gfCNCPoint3[14451] = {X 398.8006, Y 41.5563, Z -4.6667, A 0.000, B 0.000, C 0.000 }
gfCNCPoint3[14452] = {X 399.4352, Y 40.8789, Z -4.6667, A 0.000, B 0.000, C 0.000 }
gfCNCPoint3[14453] = {X 399.4352, Y 31.6953, Z -4.6667, A 0.000, B 0.000, C 0.000 }
gfCNCPoint3[14454] = {X 393.4460, Y 21.2804, Z -4.6667, A 0.000, B 0.000, C 0.000 }
gfCNCPoint3[14455] = {X 392.5594, Y 19.7721, Z -4.6667, A 0.000, B 0.000, C 0.000 }
gfCNCPoint3[14456] = {X 391.6440, Y 18.2809, Z -4.6667, A 0.000, B 0.000, C 0.000 }
gfCNCPoint3[14457] = {X 391.1727, Y 17.6249, Z -4.6667, A 0.000, B 0.000, C 0.000 }
gfCNCPoint3[14458] = {X 390.6226, Y 17.0334, Z -4.6667, A 0.000, B 0.000, C 0.000 }
gfCNCPoint3[14459] = {X 389.8677, Y 16.6248, Z -4.6667, A 0.000, B 0.000, C 0.000 }
gfCNCPoint3[14460] = {X 389.2065, Y 16.0774, Z -4.6667, A 0.000, B 0.000, C 0.000 }
gfCNCPoint3[14461] = {X 388.6642, Y 15.4120, Z -4.6667, A 0.000, B 0.000, C 0.000 }
gfCNCPoint3[14462] = {X 388.2613, Y 14.6540, Z -4.6667, A 0.000, B 0.000, C 0.000 }
gfCNCPoint3[14463] = {X 388.0133, Y 13.8322, Z -4.6667, A 0.000, B 0.000, C 0.000 }
gfCNCPoint3[14464] = {X 387.9296, Y 12.9779, Z -4.6667, A 0.000, B 0.000, C 0.000 }
gfCNCPoint3[14465] = {X 387.9296, Y 12.1868, Z -4.6667, A 0.000, B 0.000, C 0.000 }
gfCNCPoint3[14466] = {X 388.0399, Y 11.2077, Z -4.6667, A 0.000, B 0.000, C 0.000 }
gfCNCPoint3[14467] = {X 388.3654, Y 10.2777, Z -4.6667, A 0.000, B 0.000, C 0.000 }
gfCNCPoint3[14468] = {X 388.8896, Y 9.4435, Z -4.6667, A 0.000, B 0.000, C 0.000 }
gfCNCPoint3[14469] = {X 389.5863, Y 8.7468, Z -4.6667, A 0.000, B 0.000, C 0.000 }
gfCNCPoint3[14470] = {X 390.4205, Y 8.2226, Z -4.6667, A 0.000, B 0.000, C 0.000 }
gfCNCPoint3[14471] = {X 391.3505, Y 7.8971, Z -4.6667, A 0.000, B 0.000, C 0.000 }
gfCNCPoint3[14472] = {X 392.3296, Y 7.7868, Z -4.6667, A 0.000, B 0.000, C 0.000 }
gfCNCPoint3[14473] = {X 399.1118, Y 7.7868, Z -4.6667, A 0.000, B 0.000, C 0.000 }
gfCNCPoint3[14474] = {X 400.0909, Y 7.8971, Z -4.6667, A 0.000, B 0.000, C 0.000 }
gfCNCPoint3[14475] = {X 401.0208, Y 8.2226, Z -4.6667, A 0.000, B 0.000, C 0.000 }
gfCNCPoint3[14476] = {X 401.8551, Y 8.7468, Z -4.6667, A 0.000, B 0.000, C 0.000 }
gfCNCPoint3[14477] = {X 402.5518, Y 9.4435, Z -4.6667, A 0.000, B 0.000, C 0.000 }
gfCNCPoint3[14478] = {X 403.0760, Y 10.2777, Z -4.6667, A 0.000, B 0.000, C 0.000 }
gfCNCPoint3[14479] = {X 403.4014, Y 11.2077, Z -4.6667, A 0.000, B 0.000, C 0.000 }
gfCNCPoint3[14480] = {X 403.5118, Y 12.1868, Z -4.6667, A 0.000, B 0.000, C 0.000 }
gfCNCPoint3[14481] = {X 403.5115, Y 13.0233, Z -4.6667, A 0.000, B 0.000, C 0.000 }
gfCNCPoint3[14482] = {X 403.4070, Y 13.9326, Z -4.6667, A 0.000, B 0.000, C 0.000 }
gfCNCPoint3[14483] = {X 403.1165, Y 14.8007, Z -4.6667, A 0.000, B 0.000, C 0.000 }
gfCNCPoint3[14484] = {X 405.3504, Y 18.6797, Z -4.6667, A 0.000, B 0.000, C 0.000 }
gfCNCPoint3[14485] = {X 407.7810, Y 14.7428, Z -4.6667, A 0.000, B 0.000, C 0.000 }
gfCNCPoint3[14486] = {X 407.5049, Y 13.8795, Z -4.6667, A 0.000, B 0.000, C 0.000 }
gfCNCPoint3[14487] = {X 407.4115, Y 12.9779, Z -4.6667, A 0.000, B 0.000, C 0.000 }
gfCNCPoint3[14488] = {X 407.4115, Y 12.1868, Z -4.6667, A 0.000, B 0.000, C 0.000 }
gfCNCPoint3[14489] = {X 407.5219, Y 11.2077, Z -4.6667, A 0.000, B 0.000, C 0.000 }
gfCNCPoint3[14490] = {X 407.8473, Y 10.2777, Z -4.6667, A 0.000, B 0.000, C 0.000 }
gfCNCPoint3[14491] = {X 408.3715, Y 9.4435, Z -4.6667, A 0.000, B 0.000, C 0.000 }
gfCNCPoint3[14492] = {X 409.0682, Y 8.7468, Z -4.6667, A 0.000, B 0.000, C 0.000 }
gfCNCPoint3[14493] = {X 409.9025, Y 8.2226, Z -4.6667, A 0.000, B 0.000, C 0.000 }
gfCNCPoint3[14494] = {X 410.8324, Y 7.8971, Z -4.6667, A 0.000, B 0.000, C 0.000 }
gfCNCPoint3[14495] = {X 411.8115, Y 7.7868, Z -4.6667, A 0.000, B 0.000, C 0.000 }
gfCNCPoint3[14496] = {X 419.3245, Y 7.7868, Z -4.6667, A 0.000, B 0.000, C 0.000 }
gfCNCPoint3[14497] = {X 420.3036, Y 7.8971, Z -4.6667, A 0.000, B 0.000, C 0.000 }
gfCNCPoint3[14498] = {X 421.2335, Y 8.2226, Z -4.6667, A 0.000, B 0.000, C 0.000 }
gfCNCPoint3[14499] = {X 422.0678, Y 8.7468, Z -4.6667, A 0.000, B 0.000, C 0.000 }
gfCNCPoint3[14500] = {X 422.7645, Y 9.4435, Z -4.6667, A 0.000, B 0.000, C 0.000 }
gfCNCPoint3[14501] = {X 423.2887, Y 10.2777, Z -4.6667, A 0.000, B 0.000, C 0.000 }
gfCNCPoint3[14502] = {X 423.6141, Y 11.2077, Z -4.6667, A 0.000, B 0.000, C 0.000 }
gfCNCPoint3[14503] = {X 423.7245, Y 12.1868, Z -4.6667, A 0.000, B 0.000, C 0.000 }
gfCNCPoint3[14504] = {X 423.7244, Y 12.9809, Z -4.6667, A 0.000, B 0.000, C 0.000 }
gfCNCPoint3[14505] = {X 423.6306, Y 13.8597, Z -4.6667, A 0.000, B 0.000, C 0.000 }
gfCNCPoint3[14506] = {X 423.3654, Y 14.7028, Z -4.6667, A 0.000, B 0.000, C 0.000 }
gfCNCPoint3[14507] = {X 422.9393, Y 15.4771, Z -4.6667, A 0.000, B 0.000, C 0.000 }
gfCNCPoint3[14508] = {X 422.3690, Y 16.1522, Z -4.6667, A 0.000, B 0.000, C 0.000 }
gfCNCPoint3[14509] = {X 421.6768, Y 16.7018, Z -4.6667, A 0.000, B 0.000, C 0.000 }
gfCNCPoint3[14510] = {X 420.8900, Y 17.1043, Z -4.6667, A 0.000, B 0.000, C 0.000 }
gfCNCPoint3[14511] = {X 420.1830, Y 18.0570, Z -4.6667, A 0.000, B 0.000, C 0.000 }
gfCNCPoint3[14512] = {X 419.5428, Y 19.0559, Z -4.6667, A 0.000, B 0.000, C 0.000 }
gfCNCPoint3[14513] = {X 418.0618, Y 21.4538, Z -4.6667, A 0.000, B 0.000, C 0.000 }
gfCNCPoint3[14514] = {X 411.6269, Y 31.7880, Z -4.6667, A 0.000, B 0.000, C 0.000 }
gfCNCPoint3[14515] = {X 411.6276, Y 40.8617, Z -4.6667, A 0.000, B 0.000, C 0.000 }
gfCNCPoint3[14516] = {X 412.2667, Y 41.5585, Z -4.6667, A 0.000, B 0.000, C 0.000 }
gfCNCPoint3[14517] = {X 412.7469, Y 42.3730, Z -4.6667, A 0.000, B 0.000, C 0.000 }
gfCNCPoint3[14518] = {X 413.0473, Y 43.2695, Z -4.6667, A 0.000, B 0.000, C 0.000 }
gfCNCPoint3[14519] = {X 413.1547, Y 44.2089, Z -4.6667, A 0.000, B 0.000, C 0.000 }
gfCNCPoint3[14520] = {X 413.1545, Y 45.0423, Z -4.6667, A 0.000, B 0.000, C 0.000 }
gfCNCPoint3[14521] = {X 413.0719, Y 45.8494, Z -4.6667, A 0.000, B 0.000, C 0.000 }
gfCNCPoint3[14522] = {X 412.8426, Y 46.6276, Z -4.6667, A 0.000, B 0.000, C 0.000 }
gfCNCPoint3[14523] = {X 412.4743, Y 47.3505, Z -4.6667, A 0.000, B 0.000, C 0.000 }
gfCNCPoint3[14524] = {X 411.9795, Y 47.9934, Z -4.6667, A 0.000, B 0.000, C 0.000 }
gfCNCPoint3[14525] = {X 412.3313, Y 48.3200, Z -4.6667, A 0.000, B 0.000, C 0.000 }
gfCNCPoint3[14526] = {X 419.4886, Y 48.3200, Z -4.6667, A 0.000, B 0.000, C 0.000 }
gfCNCPoint3[14527] = {X 420.8006, Y 48.4093, Z -4.6667, A 0.000, B 0.000, C 0.000 }
gfCNCPoint3[14528] = {X 422.0883, Y 48.6756, Z -4.6667, A 0.000, B 0.000, C 0.000 }
gfCNCPoint3[14529] = {X 423.3281, Y 49.1140, Z -4.6667, A 0.000, B 0.000, C 0.000 }
gfCNCPoint3[14530] = {X 424.4970, Y 49.7164, Z -4.6667, A 0.000, B 0.000, C 0.000 }
gfCNCPoint3[14531] = {X 425.4625, Y 50.3832, Z -4.6667, A 0.000, B 0.000, C 0.000 }
gfCNCPoint3[14532] = {X 426.3402, Y 51.1620, Z -4.6667, A 0.000, B 0.000, C 0.000 }
gfCNCPoint3[14533] = {X 427.1172, Y 52.0412, Z -4.6667, A 0.000, B 0.000, C 0.000 }
gfCNCPoint3[14534] = {X 427.7821, Y 53.0080, Z -4.6667, A 0.000, B 0.000, C 0.000 }
gfCNCPoint3[14535] = {X 428.1267, Y 53.6313, Z -4.6667, A 0.000, B 0.000, C 0.000 }
gfCNCPoint3[14536] = {X 428.4245, Y 54.2783, Z -4.6667, A 0.000, B 0.000, C 0.000 }
gfCNCPoint3[14537] = {X 431.5824, Y 55.5088, Z -4.6667, A 0.000, B 0.000, C 0.000 }
gfCNCPoint3[14538] = {X 449.5095, Y 62.6216, Z -4.6667, A 0.000, B 0.000, C 0.000 }
gfCNCPoint3[14539] = {X 449.1114, Y 61.4466, Z -4.6667, A 0.000, B 0.000, C 0.000 }
gfCNCPoint3[14540] = {X 448.8668, Y 60.2305, Z -4.6667, A 0.000, B 0.000, C 0.000 }
gfCNCPoint3[14541] = {X 448.7798, Y 58.9930, Z -4.6667, A 0.000, B 0.000, C 0.000 }
gfCNCPoint3[14542] = {X 448.7796, Y 58.0000, Z -4.6667, A 0.000, B 0.000, C 0.000 }
gfCNCPoint3[14543] = {X 448.8564, Y 56.7833, Z -4.6667, A 0.000, B 0.000, C 0.000 }
gfCNCPoint3[14544] = {X 449.0855, Y 55.5859, Z -4.6667, A 0.000, B 0.000, C 0.000 }
gfCNCPoint3[14545] = {X 449.4632, Y 54.4268, Z -4.6667, A 0.000, B 0.000, C 0.000 }
gfCNCPoint3[14546] = {X 449.9837, Y 53.3244, Z -4.6667, A 0.000, B 0.000, C 0.000 }
gfCNCPoint3[14547] = {X 450.6386, Y 52.2961, Z -4.6667, A 0.000, B 0.000, C 0.000 }
gfCNCPoint3[14548] = {X 451.3887, Y 51.3890, Z -4.6667, A 0.000, B 0.000, C 0.000 }
gfCNCPoint3[14549] = {X 452.2434, Y 50.5796, Z -4.6667, A 0.000, B 0.000, C 0.000 }
gfCNCPoint3[14550] = {X 453.1901, Y 49.8800, Z -4.6667, A 0.000, B 0.000, C 0.000 }
gfCNCPoint3[14551] = {X 452.3731, Y 49.8442, Z -4.6667, A 0.000, B 0.000, C 0.000 }
gfCNCPoint3[14552] = {X 451.5735, Y 49.6724, Z -4.6667, A 0.000, B 0.000, C 0.000 }
gfCNCPoint3[14553] = {X 450.8138, Y 49.3696, Z -4.6667, A 0.000, B 0.000, C 0.000 }
gfCNCPoint3[14554] = {X 450.1154, Y 48.9441, Z -4.6667, A 0.000, B 0.000, C 0.000 }
gfCNCPoint3[14555] = {X 449.3503, Y 48.2496, Z -4.6667, A 0.000, B 0.000, C 0.000 }
gfCNCPoint3[14556] = {X 448.7486, Y 47.4095, Z -4.6667, A 0.000, B 0.000, C 0.000 }
gfCNCPoint3[14557] = {X 448.3373, Y 46.4616, Z -4.6667, A 0.000, B 0.000, C 0.000 }
gfCNCPoint3[14558] = {X 448.1732, Y 45.7588, Z -4.6667, A 0.000, B 0.000, C 0.000 }
gfCNCPoint3[14559] = {X 448.1146, Y 45.0395, Z -4.6667, A 0.000, B 0.000, C 0.000 }
gfCNCPoint3[14560] = {X 448.1149, Y 44.1417, Z -4.6667, A 0.000, B 0.000, C 0.000 }
gfCNCPoint3[14561] = {X 448.2252, Y 43.1751, Z -4.6667, A 0.000, B 0.000, C 0.000 }
gfCNCPoint3[14562] = {X 448.5250, Y 42.2497, Z -4.6667, A 0.000, B 0.000, C 0.000 }
gfCNCPoint3[14563] = {X 449.0024, Y 41.4021, Z -4.6667, A 0.000, B 0.000, C 0.000 }
gfCNCPoint3[14564] = {X 449.6384, Y 40.6660, Z -4.6667, A 0.000, B 0.000, C 0.000 }
gfCNCPoint3[14565] = {X 449.6384, Y 35.0338, Z -4.6667, A 0.000, B 0.000, C 0.000 }
gfCNCPoint3[14566] = {X 447.8166, Y 35.0338, Z -4.6667, A 0.000, B 0.000, C 0.000 }
gfCNCPoint3[14567] = {X 444.1904, Y 42.0943, Z -4.6667, A 0.000, B 0.000, C 0.000 }
gfCNCPoint3[14568] = {X 443.7927, Y 42.8683, Z -4.6667, A 0.000, B 0.000, C 0.000 }
gfCNCPoint3[14569] = {X 443.9302, Y 43.5105, Z -4.6667, A 0.000, B 0.000, C 0.000 }
gfCNCPoint3[14570] = {X 443.9803, Y 44.1653, Z -4.6667, A 0.000, B 0.000, C 0.000 }
gfCNCPoint3[14571] = {X 443.9805, Y 45.0000, Z -4.6667, A 0.000, B 0.000, C 0.000 }
gfCNCPoint3[14572] = {X 443.9242, Y 45.7387, Z -4.6667, A 0.000, B 0.000, C 0.000 }
gfCNCPoint3[14573] = {X 443.7568, Y 46.4603, Z -4.6667, A 0.000, B 0.000, C 0.000 }
gfCNCPoint3[14574] = {X 443.3737, Y 47.3567, Z -4.6667, A 0.000, B 0.000, C 0.000 }
gfCNCPoint3[14575] = {X 442.8199, Y 48.1591, Z -4.6667, A 0.000, B 0.000, C 0.000 }
gfCNCPoint3[14576] = {X 442.1178, Y 48.8354, Z -4.6667, A 0.000, B 0.000, C 0.000 }
gfCNCPoint3[14577] = {X 441.2952, Y 49.3586, Z -4.6667, A 0.000, B 0.000, C 0.000 }
gfCNCPoint3[14578] = {X 440.3850, Y 49.7079, Z -4.6667, A 0.000, B 0.000, C 0.000 }
gfCNCPoint3[14579] = {X 441.6485, Y 54.3386, Z -4.6667, A 0.000, B 0.000, C 0.000 }
gfCNCPoint3[14580] = {X 444.2223, Y 55.3598, Z -4.6667, A 0.000, B 0.000, C 0.000 }
gfCNCPoint3[14581] = {X 444.5426, Y 54.0016, Z -4.6667, A 0.000, B 0.000, C 0.000 }
gfCNCPoint3[14582] = {X 444.9921, Y 52.6806, Z -4.6667, A 0.000, B 0.000, C 0.000 }
gfCNCPoint3[14583] = {X 443.9523, Y 53.3763, Z -4.6667, A 0.000, B 0.000, C 0.000 }
gfCNCPoint3[14584] = {X 442.8316, Y 53.9320, Z -4.6667, A 0.000, B 0.000, C 0.000 }
gfCNCPoint3[14585] = {X 441.6485, Y 54.3386, Z -4.6667, A 0.000, B 0.000, C 0.000 }
gfCNCPoint3[14586] = {X 441.0167, Y 52.0233, Z -4.6667, A 0.000, B 0.000, C 0.000 }
gfCNCPoint3[14587] = {X 440.0672, Y 52.2155, Z -4.6667, A 0.000, B 0.000, C 0.000 }
gfCNCPoint3[14588] = {X 439.1005, Y 52.2800, Z -4.6667, A 0.000, B 0.000, C 0.000 }
gfCNCPoint3[14589] = {X 432.5144, Y 52.2800, Z -4.6667, A 0.000, B 0.000, C 0.000 }
gfCNCPoint3[14590] = {X 431.6034, Y 52.2228, Z -4.6667, A 0.000, B 0.000, C 0.000 }
gfCNCPoint3[14591] = {X 430.7067, Y 52.0520, Z -4.6667, A 0.000, B 0.000, C 0.000 }
gfCNCPoint3[14592] = {X 429.8384, Y 51.7703, Z -4.6667, A 0.000, B 0.000, C 0.000 }
gfCNCPoint3[14593] = {X 430.0169, Y 52.0771, Z -4.6667, A 0.000, B 0.000, C 0.000 }
gfCNCPoint3[14594] = {X 430.1864, Y 52.3890, Z -4.6667, A 0.000, B 0.000, C 0.000 }
gfCNCPoint3[14595] = {X 432.4641, Y 53.2767, Z -4.6667, A 0.000, B 0.000, C 0.000 }
gfCNCPoint3[14596] = {X 446.3797, Y 58.7978, Z -4.6667, A 0.000, B 0.000, C 0.000 }
gfCNCPoint3[14597] = {X 446.3796, Y 58.0000, Z -4.6667, A 0.000, B 0.000, C 0.000 }
gfCNCPoint3[14598] = {X 446.4303, Y 56.8941, Z -4.6667, A 0.000, B 0.000, C 0.000 }
gfCNCPoint3[14599] = {X 446.5821, Y 55.7974, Z -4.6667, A 0.000, B 0.000, C 0.000 }
gfCNCPoint3[14600] = {X 446.8493, Y 54.6644, Z -4.6667, A 0.000, B 0.000, C 0.000 }
gfCNCPoint3[14601] = {X 447.2243, Y 53.5622, Z -4.6667, A 0.000, B 0.000, C 0.000 }
gfCNCPoint3[14602] = {X 447.8767, Y 52.1752, Z -4.6667, A 0.000, B 0.000, C 0.000 }
gfCNCPoint3[14603] = {X 448.6995, Y 50.8820, Z -4.6667, A 0.000, B 0.000, C 0.000 }
gfCNCPoint3[14604] = {X 447.8224, Y 50.1272, Z -4.6667, A 0.000, B 0.000, C 0.000 }
gfCNCPoint3[14605] = {X 447.0760, Y 49.2431, Z -4.6667, A 0.000, B 0.000, C 0.000 }
gfCNCPoint3[14606] = {X 446.4792, Y 48.2518, Z -4.6667, A 0.000, B 0.000, C 0.000 }
gfCNCPoint3[14607] = {X 446.0469, Y 47.1785, Z -4.6667, A 0.000, B 0.000, C 0.000 }
gfCNCPoint3[14608] = {X 445.6333, Y 48.2126, Z -4.6667, A 0.000, B 0.000, C 0.000 }
gfCNCPoint3[14609] = {X 445.0668, Y 49.1715, Z -4.6667, A 0.000, B 0.000, C 0.000 }
gfCNCPoint3[14610] = {X 444.3606, Y 50.0328, Z -4.6667, A 0.000, B 0.000, C 0.000 }
gfCNCPoint3[14611] = {X 443.5314, Y 50.7763, Z -4.6667, A 0.000, B 0.000, C 0.000 }
gfCNCPoint3[14612] = {X 442.7494, Y 51.2995, Z -4.6667, A 0.000, B 0.000, C 0.000 }
gfCNCPoint3[14613] = {X 441.9065, Y 51.7175, Z -4.6667, A 0.000, B 0.000, C 0.000 }
gfCNCPoint3[14614] = {X 441.0167, Y 52.0233, Z -4.6667, A 0.000, B 0.000, C 0.000 }
gfCNCPoint3[14615] = {X 440.3850, Y 49.7079, Z -4.6667, A 0.000, B 0.000, C 0.000 }
gfCNCPoint3[14616] = {X 439.7485, Y 49.8368, Z -4.6667, A 0.000, B 0.000, C 0.000 }
gfCNCPoint3[14617] = {X 439.1005, Y 49.8800, Z -4.6667, A 0.000, B 0.000, C 0.000 }
gfCNCPoint3[14618] = {X 432.5144, Y 49.8800, Z -4.6667, A 0.000, B 0.000, C 0.000 }
gfCNCPoint3[14619] = {X 431.6014, Y 49.7938, Z -4.6667, A 0.000, B 0.000, C 0.000 }
gfCNCPoint3[14620] = {X 430.7206, Y 49.5383, Z -4.6667, A 0.000, B 0.000, C 0.000 }
gfCNCPoint3[14621] = {X 429.8343, Y 49.0782, Z -4.6667, A 0.000, B 0.000, C 0.000 }
gfCNCPoint3[14622] = {X 429.0603, Y 48.4473, Z -4.6667, A 0.000, B 0.000, C 0.000 }
gfCNCPoint3[14623] = {X 428.4309, Y 47.6720, Z -4.6667, A 0.000, B 0.000, C 0.000 }
gfCNCPoint3[14624] = {X 427.9725, Y 46.7848, Z -4.6667, A 0.000, B 0.000, C 0.000 }
gfCNCPoint3[14625] = {X 427.7197, Y 45.9083, Z -4.6667, A 0.000, B 0.000, C 0.000 }
gfCNCPoint3[14626] = {X 427.6344, Y 45.0000, Z -4.6667, A 0.000, B 0.000, C 0.000 }
gfCNCPoint3[14627] = {X 427.6344, Y 44.2089, Z -4.6667, A 0.000, B 0.000, C 0.000 }
gfCNCPoint3[14628] = {X 427.7263, Y 43.2661, Z -4.6667, A 0.000, B 0.000, C 0.000 }
gfCNCPoint3[14629] = {X 427.9987, Y 42.3588, Z -4.6667, A 0.000, B 0.000, C 0.000 }
gfCNCPoint3[14630] = {X 428.4411, Y 41.5212, Z -4.6667, A 0.000, B 0.000, C 0.000 }
gfCNCPoint3[14631] = {X 429.0371, Y 40.7849, Z -4.6667, A 0.000, B 0.000, C 0.000 }
gfCNCPoint3[14632] = {X 429.7641, Y 40.1776, Z -4.6667, A 0.000, B 0.000, C 0.000 }
gfCNCPoint3[14633] = {X 430.5947, Y 39.7222, Z -4.6667, A 0.000, B 0.000, C 0.000 }
gfCNCPoint3[14634] = {X 434.2537, Y 32.5603, Z -4.6667, A 0.000, B 0.000, C 0.000 }
gfCNCPoint3[14635] = {X 433.1657, Y 31.7642, Z -4.6667, A 0.000, B 0.000, C 0.000 }
gfCNCPoint3[14636] = {X 432.1744, Y 30.8506, Z -4.6667, A 0.000, B 0.000, C 0.000 }
gfCNCPoint3[14637] = {X 431.2923, Y 29.8311, Z -4.6667, A 0.000, B 0.000, C 0.000 }
gfCNCPoint3[14638] = {X 430.5307, Y 28.7187, Z -4.6667, A 0.000, B 0.000, C 0.000 }
gfCNCPoint3[14639] = {X 422.3160, Y 33.6865, Z -4.6667, A 0.000, B 0.000, C 0.000 }
gfCNCPoint3[14640] = {X 421.8924, Y 34.3679, Z -4.6667, A 0.000, B 0.000, C 0.000 }
gfCNCPoint3[14641] = {X 422.1472, Y 34.0999, Z -4.6667, A 0.000, B 0.000, C 0.000 }
gfCNCPoint3[14642] = {X 422.4087, Y 33.8384, Z -4.6667, A 0.000, B 0.000, C 0.000 }
gfCNCPoint3[14643] = {X 422.3622, Y 33.7626, Z -4.6667, A 0.000, B 0.000, C 0.000 }
gfCNCPoint3[14644] = {X 422.3160, Y 33.6865, Z -4.6667, A 0.000, B 0.000, C 0.000 }
gfCNCPoint3[14645] = {X 424.3697, Y 32.4446, Z -4.6667, A 0.000, B 0.000, C 0.000 }
gfCNCPoint3[14646] = {X 423.3882, Y 30.6017, Z -4.6667, A 0.000, B 0.000, C 0.000 }
gfCNCPoint3[14647] = {X 422.6133, Y 28.6629, Z -4.6667, A 0.000, B 0.000, C 0.000 }
gfCNCPoint3[14648] = {X 419.3071, Y 33.9807, Z -4.6667, A 0.000, B 0.000, C 0.000 }
gfCNCPoint3[14649] = {X 419.3074, Y 38.3388, Z -4.6667, A 0.000, B 0.000, C 0.000 }
gfCNCPoint3[14650] = {X 419.9578, Y 39.7076, Z -4.6667, A 0.000, B 0.000, C 0.000 }
gfCNCPoint3[14651] = {X 420.4336, Y 41.1465, Z -4.6667, A 0.000, B 0.000, C 0.000 }
gfCNCPoint3[14652] = {X 420.6279, Y 41.1585, Z -4.6667, A 0.000, B 0.000, C 0.000 }
gfCNCPoint3[14653] = {X 420.8222, Y 41.1728, Z -4.6667, A 0.000, B 0.000, C 0.000 }
gfCNCPoint3[14654] = {X 421.2843, Y 39.7578, Z -4.6667, A 0.000, B 0.000, C 0.000 }
gfCNCPoint3[14655] = {X 421.9170, Y 38.4105, Z -4.6667, A 0.000, B 0.000, C 0.000 }
gfCNCPoint3[14656] = {X 422.7105, Y 37.1511, Z -4.6667, A 0.000, B 0.000, C 0.000 }
gfCNCPoint3[14657] = {X 423.6530, Y 35.9990, Z -4.6667, A 0.000, B 0.000, C 0.000 }
gfCNCPoint3[14658] = {X 424.3415, Y 35.3133, Z -4.6667, A 0.000, B 0.000, C 0.000 }
gfCNCPoint3[14659] = {X 425.0829, Y 34.6852, Z -4.6667, A 0.000, B 0.000, C 0.000 }
gfCNCPoint3[14660] = {X 425.4267, Y 34.0121, Z -4.6667, A 0.000, B 0.000, C 0.000 }
gfCNCPoint3[14661] = {X 424.8788, Y 33.2414, Z -4.6667, A 0.000, B 0.000, C 0.000 }
gfCNCPoint3[14662] = {X 424.3697, Y 32.4446, Z -4.6667, A 0.000, B 0.000, C 0.000 }
gfCNCPoint3[14663] = {X 426.4233, Y 31.2026, Z -4.6667, A 0.000, B 0.000, C 0.000 }
gfCNCPoint3[14664] = {X 425.5649, Y 29.5907, Z -4.6667, A 0.000, B 0.000, C 0.000 }
gfCNCPoint3[14665] = {X 424.8871, Y 27.8950, Z -4.6667, A 0.000, B 0.000, C 0.000 }
gfCNCPoint3[14666] = {X 424.6543, Y 27.1484, Z -4.6667, A 0.000, B 0.000, C 0.000 }
gfCNCPoint3[14667] = {X 424.4565, Y 26.3919, Z -4.6667, A 0.000, B 0.000, C 0.000 }
gfCNCPoint3[14668] = {X 424.0556, Y 24.2623, Z -4.6667, A 0.000, B 0.000, C 0.000 }
gfCNCPoint3[14669] = {X 423.8652, Y 22.1037, Z -4.6667, A 0.000, B 0.000, C 0.000 }
gfCNCPoint3[14670] = {X 416.9071, Y 33.2955, Z -4.6667, A 0.000, B 0.000, C 0.000 }
gfCNCPoint3[14671] = {X 416.9075, Y 38.9954, Z -4.6667, A 0.000, B 0.000, C 0.000 }
gfCNCPoint3[14672] = {X 417.4888, Y 40.0487, Z -4.6667, A 0.000, B 0.000, C 0.000 }
gfCNCPoint3[14673] = {X 417.9368, Y 41.1651, Z -4.6667, A 0.000, B 0.000, C 0.000 }
gfCNCPoint3[14674] = {X 418.2446, Y 42.3281, Z -4.6667, A 0.000, B 0.000, C 0.000 }
gfCNCPoint3[14675] = {X 418.4076, Y 43.5200, Z -4.6667, A 0.000, B 0.000, C 0.000 }
gfCNCPoint3[14676] = {X 419.4886, Y 43.5200, Z -4.6667, A 0.000, B 0.000, C 0.000 }
gfCNCPoint3[14677] = {X 421.1752, Y 43.6186, Z -4.6667, A 0.000, B 0.000, C 0.000 }
gfCNCPoint3[14678] = {X 422.8389, Y 43.9129, Z -4.6667, A 0.000, B 0.000, C 0.000 }
gfCNCPoint3[14679] = {X 423.0005, Y 42.4234, Z -4.6667, A 0.000, B 0.000, C 0.000 }
gfCNCPoint3[14680] = {X 423.3900, Y 40.9766, Z -4.6667, A 0.000, B 0.000, C 0.000 }
gfCNCPoint3[14681] = {X 423.9980, Y 39.6073, Z -4.6667, A 0.000, B 0.000, C 0.000 }
gfCNCPoint3[14682] = {X 424.8102, Y 38.3482, Z -4.6667, A 0.000, B 0.000, C 0.000 }
gfCNCPoint3[14683] = {X 425.8068, Y 37.2295, Z -4.6667, A 0.000, B 0.000, C 0.000 }
gfCNCPoint3[14684] = {X 426.9642, Y 36.2780, Z -4.6667, A 0.000, B 0.000, C 0.000 }
gfCNCPoint3[14685] = {X 428.2773, Y 33.7078, Z -4.6667, A 0.000, B 0.000, C 0.000 }
gfCNCPoint3[14686] = {X 427.2919, Y 32.4984, Z -4.6667, A 0.000, B 0.000, C 0.000 }
gfCNCPoint3[14687] = {X 426.4233, Y 31.2026, Z -4.6667, A 0.000, B 0.000, C 0.000 }
gfCNCPoint3[14688] = {X 428.4770, Y 29.9607, Z -4.6667, A 0.000, B 0.000, C 0.000 }
gfCNCPoint3[14689] = {X 427.7729, Y 28.6468, Z -4.6667, A 0.000, B 0.000, C 0.000 }
gfCNCPoint3[14690] = {X 427.2090, Y 27.2670, Z -4.6667, A 0.000, B 0.000, C 0.000 }
gfCNCPoint3[14691] = {X 426.7913, Y 25.8360, Z -4.6667, A 0.000, B 0.000, C 0.000 }
gfCNCPoint3[14692] = {X 426.4333, Y 23.9362, Z -4.6667, A 0.000, B 0.000, C 0.000 }
gfCNCPoint3[14693] = {X 426.2634, Y 22.0104, Z -4.6667, A 0.000, B 0.000, C 0.000 }
gfCNCPoint3[14694] = {X 426.2915, Y 19.9433, Z -4.6667, A 0.000, B 0.000, C 0.000 }
gfCNCPoint3[14695] = {X 426.5362, Y 17.8906, Z -4.6667, A 0.000, B 0.000, C 0.000 }
gfCNCPoint3[14696] = {X 426.9947, Y 15.8749, Z -4.6667, A 0.000, B 0.000, C 0.000 }
gfCNCPoint3[14697] = {X 427.6132, Y 14.1191, Z -4.6667, A 0.000, B 0.000, C 0.000 }
gfCNCPoint3[14698] = {X 428.4475, Y 12.4549, Z -4.6667, A 0.000, B 0.000, C 0.000 }
gfCNCPoint3[14699] = {X 429.4841, Y 10.9087, Z -4.6667, A 0.000, B 0.000, C 0.000 }
gfCNCPoint3[14700] = {X 430.7069, Y 9.5050, Z -4.6667, A 0.000, B 0.000, C 0.000 }
gfCNCPoint3[14701] = {X 426.0925, Y 9.5050, Z -4.6667, A 0.000, B 0.000, C 0.000 }
gfCNCPoint3[14702] = {X 426.3754, Y 10.3750, Z -4.6667, A 0.000, B 0.000, C 0.000 }
gfCNCPoint3[14703] = {X 426.5470, Y 11.2737, Z -4.6667, A 0.000, B 0.000, C 0.000 }
gfCNCPoint3[14704] = {X 426.6045, Y 12.1868, Z -4.6667, A 0.000, B 0.000, C 0.000 }
gfCNCPoint3[14705] = {X 426.6045, Y 12.9851, Z -4.6667, A 0.000, B 0.000, C 0.000 }
gfCNCPoint3[14706] = {X 426.4815, Y 14.2871, Z -4.6667, A 0.000, B 0.000, C 0.000 }
gfCNCPoint3[14707] = {X 426.1296, Y 15.5465, Z -4.6667, A 0.000, B 0.000, C 0.000 }
gfCNCPoint3[14708] = {X 425.5599, Y 16.7236, Z -4.6667, A 0.000, B 0.000, C 0.000 }
gfCNCPoint3[14709] = {X 424.7904, Y 17.7810, Z -4.6667, A 0.000, B 0.000, C 0.000 }
gfCNCPoint3[14710] = {X 423.8456, Y 18.6852, Z -4.6667, A 0.000, B 0.000, C 0.000 }
gfCNCPoint3[14711] = {X 422.7555, Y 19.4074, Z -4.6667, A 0.000, B 0.000, C 0.000 }
gfCNCPoint3[14712] = {X 422.3655, Y 19.9717, Z -4.6667, A 0.000, B 0.000, C 0.000 }
gfCNCPoint3[14713] = {X 422.0027, Y 20.5539, Z -4.6667, A 0.000, B 0.000, C 0.000 }
gfCNCPoint3[14714] = {X 414.5070, Y 32.6104, Z -4.6667, A 0.000, B 0.000, C 0.000 }
gfCNCPoint3[14715] = {X 414.5075, Y 39.7469, Z -4.6667, A 0.000, B 0.000, C 0.000 }
gfCNCPoint3[14716] = {X 415.1561, Y 40.7519, Z -4.6667, A 0.000, B 0.000, C 0.000 }
gfCNCPoint3[14717] = {X 415.6344, Y 41.8483, Z -4.6667, A 0.000, B 0.000, C 0.000 }
gfCNCPoint3[14718] = {X 415.9298, Y 43.0074, Z -4.6667, A 0.000, B 0.000, C 0.000 }
gfCNCPoint3[14719] = {X 416.0347, Y 44.1990, Z -4.6667, A 0.000, B 0.000, C 0.000 }
gfCNCPoint3[14720] = {X 416.0347, Y 44.9999, Z -4.6667, A 0.000, B 0.000, C 0.000 }
gfCNCPoint3[14721] = {X 416.0201, Y 45.4609, Z -4.6667, A 0.000, B 0.000, C 0.000 }
gfCNCPoint3[14722] = {X 415.9763, Y 45.9200, Z -4.6667, A 0.000, B 0.000, C 0.000 }
gfCNCPoint3[14723] = {X 419.4886, Y 45.9200, Z -4.6667, A 0.000, B 0.000, C 0.000 }
gfCNCPoint3[14724] = {X 420.8957, Y 46.0022, Z -4.6667, A 0.000, B 0.000, C 0.000 }
gfCNCPoint3[14725] = {X 422.2836, Y 46.2478, Z -4.6667, A 0.000, B 0.000, C 0.000 }
gfCNCPoint3[14726] = {X 423.4822, Y 46.5992, Z -4.6667, A 0.000, B 0.000, C 0.000 }
gfCNCPoint3[14727] = {X 424.6380, Y 47.0725, Z -4.6667, A 0.000, B 0.000, C 0.000 }
gfCNCPoint3[14728] = {X 425.7388, Y 47.6626, Z -4.6667, A 0.000, B 0.000, C 0.000 }
gfCNCPoint3[14729] = {X 425.4600, Y 46.7984, Z -4.6667, A 0.000, B 0.000, C 0.000 }
gfCNCPoint3[14730] = {X 425.2910, Y 45.9063, Z -4.6667, A 0.000, B 0.000, C 0.000 }
gfCNCPoint3[14731] = {X 425.2344, Y 45.0000, Z -4.6667, A 0.000, B 0.000, C 0.000 }
gfCNCPoint3[14732] = {X 425.2344, Y 44.2089, Z -4.6667, A 0.000, B 0.000, C 0.000 }
gfCNCPoint3[14733] = {X 425.2353, Y 44.0976, Z -4.6667, A 0.000, B 0.000, C 0.000 }
gfCNCPoint3[14734] = {X 425.2378, Y 43.9863, Z -4.6667, A 0.000, B 0.000, C 0.000 }
gfCNCPoint3[14735] = {X 425.3770, Y 42.7748, Z -4.6667, A 0.000, B 0.000, C 0.000 }
gfCNCPoint3[14736] = {X 425.7165, Y 41.6036, Z -4.6667, A 0.000, B 0.000, C 0.000 }
gfCNCPoint3[14737] = {X 426.2468, Y 40.5054, Z -4.6667, A 0.000, B 0.000, C 0.000 }
gfCNCPoint3[14738] = {X 426.9528, Y 39.5112, Z -4.6667, A 0.000, B 0.000, C 0.000 }
gfCNCPoint3[14739] = {X 427.8150, Y 38.6488, Z -4.6667, A 0.000, B 0.000, C 0.000 }
gfCNCPoint3[14740] = {X 428.8090, Y 37.9424, Z -4.6667, A 0.000, B 0.000, C 0.000 }
gfCNCPoint3[14741] = {X 431.2079, Y 33.2468, Z -4.6667, A 0.000, B 0.000, C 0.000 }
gfCNCPoint3[14742] = {X 430.1898, Y 32.2441, Z -4.6667, A 0.000, B 0.000, C 0.000 }
gfCNCPoint3[14743] = {X 429.2764, Y 31.1451, Z -4.6667, A 0.000, B 0.000, C 0.000 }
gfCNCPoint3[14744] = {X 428.4770, Y 29.9607, Z -4.6667, A 0.000, B 0.000, C 0.000 }
gfCNCPoint3[14745] = {X 430.5307, Y 28.7187, Z -4.6667, A 0.000, B 0.000, C 0.000 }
gfCNCPoint3[14746] = {X 429.9438, Y 27.6235, Z -4.6667, A 0.000, B 0.000, C 0.000 }
gfCNCPoint3[14747] = {X 429.4739, Y 26.4732, Z -4.6667, A 0.000, B 0.000, C 0.000 }
gfCNCPoint3[14748] = {X 429.1261, Y 25.2803, Z -4.6667, A 0.000, B 0.000, C 0.000 }
gfCNCPoint3[14749] = {X 428.8017, Y 23.5412, Z -4.6667, A 0.000, B 0.000, C 0.000 }
gfCNCPoint3[14750] = {X 428.6567, Y 21.7780, Z -4.6667, A 0.000, B 0.000, C 0.000 }
gfCNCPoint3[14751] = {X 428.6927, Y 20.0093, Z -4.6667, A 0.000, B 0.000, C 0.000 }
gfCNCPoint3[14752] = {X 428.9091, Y 18.2534, Z -4.6667, A 0.000, B 0.000, C 0.000 }
gfCNCPoint3[14753] = {X 429.3039, Y 16.5289, Z -4.6667, A 0.000, B 0.000, C 0.000 }
gfCNCPoint3[14754] = {X 429.8220, Y 15.0579, Z -4.6667, A 0.000, B 0.000, C 0.000 }
gfCNCPoint3[14755] = {X 430.5209, Y 13.6636, Z -4.6667, A 0.000, B 0.000, C 0.000 }
gfCNCPoint3[14756] = {X 431.3894, Y 12.3682, Z -4.6667, A 0.000, B 0.000, C 0.000 }
gfCNCPoint3[14757] = {X 432.4138, Y 11.1921, Z -4.6667, A 0.000, B 0.000, C 0.000 }
gfCNCPoint3[14758] = {X 433.5453, Y 10.1797, Z -4.6667, A 0.000, B 0.000, C 0.000 }
gfCNCPoint3[14759] = {X 434.7922, Y 9.3133, Z -4.6667, A 0.000, B 0.000, C 0.000 }
gfCNCPoint3[14760] = {X 436.1357, Y 8.6059, Z -4.6667, A 0.000, B 0.000, C 0.000 }
gfCNCPoint3[14761] = {X 437.5557, Y 8.0683, Z -4.6667, A 0.000, B 0.000, C 0.000 }
gfCNCPoint3[14762] = {X 439.0307, Y 7.7083, Z -4.6667, A 0.000, B 0.000, C 0.000 }
gfCNCPoint3[14763] = {X 441.1775, Y 7.4110, Z -4.6667, A 0.000, B 0.000, C 0.000 }
gfCNCPoint3[14764] = {X 443.3425, Y 7.3146, Z -4.6667, A 0.000, B 0.000, C 0.000 }
gfCNCPoint3[14765] = {X 459.4467, Y 7.3106, Z -4.6667, A 0.000, B 0.000, C 0.000 }
gfCNCPoint3[14766] = {X 460.4095, Y 7.4067, Z -4.6667, A 0.000, B 0.000, C 0.000 }
gfCNCPoint3[14767] = {X 461.3344, Y 7.6912, Z -4.6667, A 0.000, B 0.000, C 0.000 }
gfCNCPoint3[14768] = {X 462.1847, Y 8.1529, Z -4.6667, A 0.000, B 0.000, C 0.000 }
gfCNCPoint3[14769] = {X 462.9270, Y 8.7735, Z -4.6667, A 0.000, B 0.000, C 0.000 }
gfCNCPoint3[14770] = {X 463.5320, Y 9.5287, Z -4.6667, A 0.000, B 0.000, C 0.000 }
gfCNCPoint3[14771] = {X 463.9758, Y 10.3885, Z -4.6667, A 0.000, B 0.000, C 0.000 }
gfCNCPoint3[14772] = {X 464.2317, Y 11.2690, Z -4.6667, A 0.000, B 0.000, C 0.000 }
gfCNCPoint3[14773] = {X 464.3179, Y 12.1818, Z -4.6667, A 0.000, B 0.000, C 0.000 }
gfCNCPoint3[14774] = {X 464.3179, Y 12.9780, Z -4.6667, A 0.000, B 0.000, C 0.000 }
gfCNCPoint3[14775] = {X 464.2174, Y 13.9636, Z -4.6667, A 0.000, B 0.000, C 0.000 }
gfCNCPoint3[14776] = {X 463.9198, Y 14.9087, Z -4.6667, A 0.000, B 0.000, C 0.000 }
gfCNCPoint3[14777] = {X 463.4375, Y 15.7741, Z -4.6667, A 0.000, B 0.000, C 0.000 }
gfCNCPoint3[14778] = {X 462.7903, Y 16.5243, Z -4.6667, A 0.000, B 0.000, C 0.000 }
gfCNCPoint3[14779] = {X 462.7900, Y 16.7697, Z -4.6667, A 0.000, B 0.000, C 0.000 }
gfCNCPoint3[14780] = {X 462.7910, Y 40.6632, Z -4.6667, A 0.000, B 0.000, C 0.000 }
gfCNCPoint3[14781] = {X 463.4319, Y 41.4048, Z -4.6667, A 0.000, B 0.000, C 0.000 }
gfCNCPoint3[14782] = {X 463.9117, Y 42.2594, Z -4.6667, A 0.000, B 0.000, C 0.000 }
gfCNCPoint3[14783] = {X 464.2110, Y 43.1927, Z -4.6667, A 0.000, B 0.000, C 0.000 }
gfCNCPoint3[14784] = {X 464.3178, Y 44.1670, Z -4.6667, A 0.000, B 0.000, C 0.000 }
gfCNCPoint3[14785] = {X 464.3179, Y 45.0000, Z -4.6667, A 0.000, B 0.000, C 0.000 }
gfCNCPoint3[14786] = {X 464.3081, Y 45.3090, Z -4.6667, A 0.000, B 0.000, C 0.000 }
gfCNCPoint3[14787] = {X 464.2788, Y 45.6167, Z -4.6667, A 0.000, B 0.000, C 0.000 }
gfCNCPoint3[14788] = {X 464.0485, Y 46.5992, Z -4.6667, A 0.000, B 0.000, C 0.000 }
gfCNCPoint3[14789] = {X 463.6209, Y 47.5134, Z -4.6667, A 0.000, B 0.000, C 0.000 }
gfCNCPoint3[14790] = {X 463.0145, Y 48.3200, Z -4.6667, A 0.000, B 0.000, C 0.000 }
gfCNCPoint3[14791] = {X 462.6627, Y 47.9934, Z -4.6667, A 0.000, B 0.000, C 0.000 }
gfCNCPoint3[14792] = {X 461.9835, Y 48.5889, Z -4.6667, A 0.000, B 0.000, C 0.000 }
gfCNCPoint3[14793] = {X 461.1970, Y 49.0331, Z -4.6667, A 0.000, B 0.000, C 0.000 }
gfCNCPoint3[14794] = {X 460.3364, Y 49.3073, Z -4.6667, A 0.000, B 0.000, C 0.000 }
gfCNCPoint3[14795] = {X 459.4379, Y 49.4000, Z -4.6667, A 0.000, B 0.000, C 0.000 }
gfCNCPoint3[14796] = {X 452.9945, Y 49.4000, Z -4.6667, A 0.000, B 0.000, C 0.000 }
gfCNCPoint3[14797] = {X 452.0154, Y 49.2897, Z -4.6667, A 0.000, B 0.000, C 0.000 }
gfCNCPoint3[14798] = {X 451.0854, Y 48.9643, Z -4.6667, A 0.000, B 0.000, C 0.000 }
gfCNCPoint3[14799] = {X 450.2511, Y 48.4400, Z -4.6667, A 0.000, B 0.000, C 0.000 }
gfCNCPoint3[14800] = {X 449.5544, Y 47.7433, Z -4.6667, A 0.000, B 0.000, C 0.000 }
gfCNCPoint3[14801] = {X 449.0302, Y 46.9091, Z -4.6667, A 0.000, B 0.000, C 0.000 }
gfCNCPoint3[14802] = {X 448.7048, Y 45.9791, Z -4.6667, A 0.000, B 0.000, C 0.000 }
gfCNCPoint3[14803] = {X 448.5945, Y 45.0000, Z -4.6667, A 0.000, B 0.000, C 0.000 }
gfCNCPoint3[14804] = {X 448.5949, Y 44.1483, Z -4.6667, A 0.000, B 0.000, C 0.000 }
gfCNCPoint3[14805] = {X 448.7053, Y 43.2275, Z -4.6667, A 0.000, B 0.000, C 0.000 }
gfCNCPoint3[14806] = {X 449.0063, Y 42.3503, Z -4.6667, A 0.000, B 0.000, C 0.000 }
gfCNCPoint3[14807] = {X 449.4844, Y 41.5556, Z -4.6667, A 0.000, B 0.000, C 0.000 }
gfCNCPoint3[14808] = {X 450.1184, Y 40.8789, Z -4.6667, A 0.000, B 0.000, C 0.000 }
gfCNCPoint3[14809] = {X 450.1184, Y 34.5538, Z -4.6667, A 0.000, B 0.000, C 0.000 }
gfCNCPoint3[14810] = {X 447.5235, Y 34.5538, Z -4.6667, A 0.000, B 0.000, C 0.000 }
gfCNCPoint3[14811] = {X 443.7635, Y 41.8750, Z -4.6667, A 0.000, B 0.000, C 0.000 }
gfCNCPoint3[14812] = {X 443.2765, Y 42.8228, Z -4.6667, A 0.000, B 0.000, C 0.000 }
gfCNCPoint3[14813] = {X 443.4441, Y 43.5069, Z -4.6667, A 0.000, B 0.000, C 0.000 }
gfCNCPoint3[14814] = {X 443.5005, Y 44.2089, Z -4.6667, A 0.000, B 0.000, C 0.000 }
gfCNCPoint3[14815] = {X 443.5005, Y 45.0000, Z -4.6667, A 0.000, B 0.000, C 0.000 }
gfCNCPoint3[14816] = {X 443.3902, Y 45.9791, Z -4.6667, A 0.000, B 0.000, C 0.000 }
gfCNCPoint3[14817] = {X 443.0647, Y 46.9091, Z -4.6667, A 0.000, B 0.000, C 0.000 }
gfCNCPoint3[14818] = {X 442.5405, Y 47.7434, Z -4.6667, A 0.000, B 0.000, C 0.000 }
gfCNCPoint3[14819] = {X 441.8438, Y 48.4401, Z -4.6667, A 0.000, B 0.000, C 0.000 }
gfCNCPoint3[14820] = {X 441.0096, Y 48.9643, Z -4.6667, A 0.000, B 0.000, C 0.000 }
gfCNCPoint3[14821] = {X 440.0796, Y 49.2897, Z -4.6667, A 0.000, B 0.000, C 0.000 }
gfCNCPoint3[14822] = {X 439.1005, Y 49.4000, Z -4.6667, A 0.000, B 0.000, C 0.000 }
gfCNCPoint3[14823] = {X 432.5144, Y 49.4000, Z -4.6667, A 0.000, B 0.000, C 0.000 }
gfCNCPoint3[14824] = {X 431.5353, Y 49.2897, Z -4.6667, A 0.000, B 0.000, C 0.000 }
gfCNCPoint3[14825] = {X 430.6053, Y 48.9643, Z -4.6667, A 0.000, B 0.000, C 0.000 }
gfCNCPoint3[14826] = {X 429.7711, Y 48.4401, Z -4.6667, A 0.000, B 0.000, C 0.000 }
gfCNCPoint3[14827] = {X 429.0743, Y 47.7434, Z -4.6667, A 0.000, B 0.000, C 0.000 }
gfCNCPoint3[14828] = {X 428.5501, Y 46.9091, Z -4.6667, A 0.000, B 0.000, C 0.000 }
gfCNCPoint3[14829] = {X 428.2247, Y 45.9791, Z -4.6667, A 0.000, B 0.000, C 0.000 }
gfCNCPoint3[14830] = {X 428.1144, Y 45.0000, Z -4.6667, A 0.000, B 0.000, C 0.000 }
gfCNCPoint3[14831] = {X 428.1148, Y 44.1483, Z -4.6667, A 0.000, B 0.000, C 0.000 }
gfCNCPoint3[14832] = {X 428.2132, Y 43.2816, Z -4.6667, A 0.000, B 0.000, C 0.000 }
gfCNCPoint3[14833] = {X 428.4806, Y 42.4514, Z -4.6667, A 0.000, B 0.000, C 0.000 }
gfCNCPoint3[14834] = {X 428.9065, Y 41.6903, Z -4.6667, A 0.000, B 0.000, C 0.000 }
gfCNCPoint3[14835] = {X 429.4741, Y 41.0281, Z -4.6667, A 0.000, B 0.000, C 0.000 }
gfCNCPoint3[14836] = {X 430.1613, Y 40.4909, Z -4.6667, A 0.000, B 0.000, C 0.000 }
gfCNCPoint3[14837] = {X 430.9408, Y 40.0998, Z -4.6667, A 0.000, B 0.000, C 0.000 }
gfCNCPoint3[14838] = {X 434.8818, Y 32.3858, Z -4.6667, A 0.000, B 0.000, C 0.000 }
gfCNCPoint3[14839] = {X 433.6222, Y 31.5160, Z -4.6667, A 0.000, B 0.000, C 0.000 }
gfCNCPoint3[14840] = {X 432.4897, Y 30.4861, Z -4.6667, A 0.000, B 0.000, C 0.000 }
gfCNCPoint3[14841] = {X 431.5045, Y 29.3146, Z -4.6667, A 0.000, B 0.000, C 0.000 }
gfCNCPoint3[14842] = {X 430.6841, Y 28.0223, Z -4.6667, A 0.000, B 0.000, C 0.000 }
gfCNCPoint3[14843] = {X 430.0431, Y 26.6322, Z -4.6667, A 0.000, B 0.000, C 0.000 }
gfCNCPoint3[14844] = {X 429.5930, Y 25.1691, Z -4.6667, A 0.000, B 0.000, C 0.000 }
gfCNCPoint3[14845] = {X 429.2775, Y 23.4781, Z -4.6667, A 0.000, B 0.000, C 0.000 }
gfCNCPoint3[14846] = {X 429.1365, Y 21.7637, Z -4.6667, A 0.000, B 0.000, C 0.000 }
gfCNCPoint3[14847] = {X 429.1714, Y 20.0439, Z -4.6667, A 0.000, B 0.000, C 0.000 }
gfCNCPoint3[14848] = {X 429.3819, Y 18.3366, Z -4.6667, A 0.000, B 0.000, C 0.000 }
gfCNCPoint3[14849] = {X 429.7657, Y 16.6598, Z -4.6667, A 0.000, B 0.000, C 0.000 }
gfCNCPoint3[14850] = {X 430.3284, Y 15.0962, Z -4.6667, A 0.000, B 0.000, C 0.000 }
gfCNCPoint3[14851] = {X 431.1033, Y 13.6263, Z -4.6667, A 0.000, B 0.000, C 0.000 }
gfCNCPoint3[14852] = {X 432.0753, Y 12.2785, Z -4.6667, A 0.000, B 0.000, C 0.000 }
gfCNCPoint3[14853] = {X 433.2255, Y 11.0791, Z -4.6667, A 0.000, B 0.000, C 0.000 }
gfCNCPoint3[14854] = {X 434.5314, Y 10.0515, Z -4.6667, A 0.000, B 0.000, C 0.000 }
gfCNCPoint3[14855] = {X 435.9676, Y 9.2157, Z -4.6667, A 0.000, B 0.000, C 0.000 }
gfCNCPoint3[14856] = {X 437.5062, Y 8.5879, Z -4.6667, A 0.000, B 0.000, C 0.000 }
gfCNCPoint3[14857] = {X 439.1172, Y 8.1805, Z -4.6667, A 0.000, B 0.000, C 0.000 }
gfCNCPoint3[14858] = {X 441.2213, Y 7.8890, Z -4.6667, A 0.000, B 0.000, C 0.000 }
gfCNCPoint3[14859] = {X 443.3434, Y 7.7946, Z -4.6667, A 0.000, B 0.000, C 0.000 }
gfCNCPoint3[14860] = {X 444.0367, Y 7.7906, Z -4.6667, A 0.000, B 0.000, C 0.000 }
gfCNCPoint3[14861] = {X 459.4467, Y 7.7906, Z -4.6667, A 0.000, B 0.000, C 0.000 }
gfCNCPoint3[14862] = {X 460.4239, Y 7.9007, Z -4.6667, A 0.000, B 0.000, C 0.000 }
gfCNCPoint3[14863] = {X 461.3520, Y 8.2254, Z -4.6667, A 0.000, B 0.000, C 0.000 }
gfCNCPoint3[14864] = {X 462.1846, Y 8.7486, Z -4.6667, A 0.000, B 0.000, C 0.000 }
gfCNCPoint3[14865] = {X 462.8799, Y 9.4439, Z -4.6667, A 0.000, B 0.000, C 0.000 }
gfCNCPoint3[14866] = {X 463.4031, Y 10.2765, Z -4.6667, A 0.000, B 0.000, C 0.000 }
gfCNCPoint3[14867] = {X 463.7278, Y 11.2047, Z -4.6667, A 0.000, B 0.000, C 0.000 }
gfCNCPoint3[14868] = {X 463.8379, Y 12.1818, Z -4.6667, A 0.000, B 0.000, C 0.000 }
gfCNCPoint3[14869] = {X 463.8377, Y 13.0201, Z -4.6667, A 0.000, B 0.000, C 0.000 }
gfCNCPoint3[14870] = {X 463.7299, Y 13.9470, Z -4.6667, A 0.000, B 0.000, C 0.000 }
gfCNCPoint3[14871] = {X 463.4291, Y 14.8303, Z -4.6667, A 0.000, B 0.000, C 0.000 }
gfCNCPoint3[14872] = {X 462.9487, Y 15.6303, Z -4.6667, A 0.000, B 0.000, C 0.000 }
gfCNCPoint3[14873] = {X 462.3105, Y 16.3110, Z -4.6667, A 0.000, B 0.000, C 0.000 }
gfCNCPoint3[14874] = {X 462.3100, Y 16.7692, Z -4.6667, A 0.000, B 0.000, C 0.000 }
gfCNCPoint3[14875] = {X 462.3110, Y 40.8763, Z -4.6667, A 0.000, B 0.000, C 0.000 }
gfCNCPoint3[14876] = {X 462.9554, Y 41.5654, Z -4.6667, A 0.000, B 0.000, C 0.000 }
gfCNCPoint3[14877] = {X 463.4381, Y 42.3760, Z -4.6667, A 0.000, B 0.000, C 0.000 }
gfCNCPoint3[14878] = {X 463.7368, Y 43.2709, Z -4.6667, A 0.000, B 0.000, C 0.000 }
gfCNCPoint3[14879] = {X 463.8379, Y 44.2089, Z -4.6667, A 0.000, B 0.000, C 0.000 }
gfCNCPoint3[14880] = {X 463.8379, Y 45.0000, Z -4.6667, A 0.000, B 0.000, C 0.000 }
gfCNCPoint3[14881] = {X 463.7612, Y 45.8182, Z -4.6667, A 0.000, B 0.000, C 0.000 }
gfCNCPoint3[14882] = {X 463.5336, Y 46.6079, Z -4.6667, A 0.000, B 0.000, C 0.000 }
gfCNCPoint3[14883] = {X 463.1632, Y 47.3415, Z -4.6667, A 0.000, B 0.000, C 0.000 }
gfCNCPoint3[14884] = {X 462.6627, Y 47.9934, Z -4.6667, A 0.000, B 0.000, C 0.000 }
gfCNCPoint3[14885] = {X 463.0145, Y 48.3200, Z -4.6667, A 0.000, B 0.000, C 0.000 }
gfCNCPoint3[14886] = {X 472.1884, Y 48.3200, Z -4.6667, A 0.000, B 0.000, C 0.000 }
gfCNCPoint3[14887] = {X 471.5820, Y 47.5134, Z -4.6667, A 0.000, B 0.000, C 0.000 }
gfCNCPoint3[14888] = {X 471.1544, Y 46.5992, Z -4.6667, A 0.000, B 0.000, C 0.000 }
gfCNCPoint3[14889] = {X 470.9241, Y 45.6167, Z -4.6667, A 0.000, B 0.000, C 0.000 }
gfCNCPoint3[14890] = {X 470.8947, Y 45.3090, Z -4.6667, A 0.000, B 0.000, C 0.000 }
gfCNCPoint3[14891] = {X 470.8850, Y 45.0000, Z -4.6667, A 0.000, B 0.000, C 0.000 }
gfCNCPoint3[14892] = {X 470.8850, Y 44.2089, Z -4.6667, A 0.000, B 0.000, C 0.000 }
gfCNCPoint3[14893] = {X 470.9769, Y 43.2661, Z -4.6667, A 0.000, B 0.000, C 0.000 }
gfCNCPoint3[14894] = {X 471.2492, Y 42.3588, Z -4.6667, A 0.000, B 0.000, C 0.000 }
gfCNCPoint3[14895] = {X 471.6917, Y 41.5212, Z -4.6667, A 0.000, B 0.000, C 0.000 }
gfCNCPoint3[14896] = {X 472.2877, Y 40.7849, Z -4.6667, A 0.000, B 0.000, C 0.000 }
gfCNCPoint3[14897] = {X 473.0147, Y 40.1776, Z -4.6667, A 0.000, B 0.000, C 0.000 }
gfCNCPoint3[14898] = {X 473.8453, Y 39.7222, Z -4.6667, A 0.000, B 0.000, C 0.000 }
gfCNCPoint3[14899] = {X 477.5003, Y 32.5679, Z -4.6667, A 0.000, B 0.000, C 0.000 }
gfCNCPoint3[14900] = {X 476.2830, Y 31.6579, Z -4.6667, A 0.000, B 0.000, C 0.000 }
gfCNCPoint3[14901] = {X 475.1902, Y 30.6018, Z -4.6667, A 0.000, B 0.000, C 0.000 }
gfCNCPoint3[14902] = {X 474.2392, Y 29.4163, Z -4.6667, A 0.000, B 0.000, C 0.000 }
gfCNCPoint3[14903] = {X 473.4454, Y 28.1203, Z -4.6667, A 0.000, B 0.000, C 0.000 }
gfCNCPoint3[14904] = {X 472.8212, Y 26.7346, Z -4.6667, A 0.000, B 0.000, C 0.000 }
gfCNCPoint3[14905] = {X 472.3768, Y 25.2812, Z -4.6667, A 0.000, B 0.000, C 0.000 }
gfCNCPoint3[14906] = {X 472.0521, Y 23.5419, Z -4.6667, A 0.000, B 0.000, C 0.000 }
gfCNCPoint3[14907] = {X 471.9069, Y 21.7785, Z -4.6667, A 0.000, B 0.000, C 0.000 }
gfCNCPoint3[14908] = {X 471.9428, Y 20.0095, Z -4.6667, A 0.000, B 0.000, C 0.000 }
gfCNCPoint3[14909] = {X 472.1594, Y 18.2535, Z -4.6667, A 0.000, B 0.000, C 0.000 }
gfCNCPoint3[14910] = {X 472.5544, Y 16.5288, Z -4.6667, A 0.000, B 0.000, C 0.000 }
gfCNCPoint3[14911] = {X 473.0730, Y 15.0578, Z -4.6667, A 0.000, B 0.000, C 0.000 }
gfCNCPoint3[14912] = {X 473.7723, Y 13.6637, Z -4.6667, A 0.000, B 0.000, C 0.000 }
gfCNCPoint3[14913] = {X 474.6412, Y 12.3684, Z -4.6667, A 0.000, B 0.000, C 0.000 }
gfCNCPoint3[14914] = {X 475.6660, Y 11.1925, Z -4.6667, A 0.000, B 0.000, C 0.000 }
gfCNCPoint3[14915] = {X 476.7435, Y 10.2235, Z -4.6667, A 0.000, B 0.000, C 0.000 }
gfCNCPoint3[14916] = {X 477.9269, Y 9.3868, Z -4.6667, A 0.000, B 0.000, C 0.000 }
gfCNCPoint3[14917] = {X 479.1998, Y 8.6940, Z -4.6667, A 0.000, B 0.000, C 0.000 }
gfCNCPoint3[14918] = {X 480.5449, Y 8.1546, Z -4.6667, A 0.000, B 0.000, C 0.000 }
gfCNCPoint3[14919] = {X 481.9438, Y 7.7760, Z -4.6667, A 0.000, B 0.000, C 0.000 }
gfCNCPoint3[14920] = {X 484.0949, Y 7.4406, Z -4.6667, A 0.000, B 0.000, C 0.000 }
gfCNCPoint3[14921] = {X 486.2688, Y 7.3228, Z -4.6667, A 0.000, B 0.000, C 0.000 }
gfCNCPoint3[14922] = {X 486.9707, Y 7.3106, Z -4.6667, A 0.000, B 0.000, C 0.000 }
gfCNCPoint3[14923] = {X 502.2122, Y 7.3106, Z -4.6667, A 0.000, B 0.000, C 0.000 }
gfCNCPoint3[14924] = {X 502.7438, Y 7.3147, Z -4.6667, A 0.000, B 0.000, C 0.000 }
gfCNCPoint3[14925] = {X 503.6981, Y 7.4169, Z -4.6667, A 0.000, B 0.000, C 0.000 }
gfCNCPoint3[14926] = {X 504.6138, Y 7.7045, Z -4.6667, A 0.000, B 0.000, C 0.000 }
gfCNCPoint3[14927] = {X 505.4551, Y 8.1664, Z -4.6667, A 0.000, B 0.000, C 0.000 }
gfCNCPoint3[14928] = {X 506.1893, Y 8.7845, Z -4.6667, A 0.000, B 0.000, C 0.000 }
gfCNCPoint3[14929] = {X 506.7879, Y 9.5348, Z -4.6667, A 0.000, B 0.000, C 0.000 }
gfCNCPoint3[14930] = {X 507.2274, Y 10.3880, Z -4.6667, A 0.000, B 0.000, C 0.000 }
gfCNCPoint3[14931] = {X 507.4824, Y 11.2665, Z -4.6667, A 0.000, B 0.000, C 0.000 }
gfCNCPoint3[14932] = {X 507.5685, Y 12.1773, Z -4.6667, A 0.000, B 0.000, C 0.000 }
gfCNCPoint3[14933] = {X 507.5683, Y 13.0237, Z -4.6667, A 0.000, B 0.000, C 0.000 }
gfCNCPoint3[14934] = {X 507.4609, Y 13.9971, Z -4.6667, A 0.000, B 0.000, C 0.000 }
gfCNCPoint3[14935] = {X 507.1613, Y 14.9294, Z -4.6667, A 0.000, B 0.000, C 0.000 }
gfCNCPoint3[14936] = {X 506.6817, Y 15.7832, Z -4.6667, A 0.000, B 0.000, C 0.000 }
gfCNCPoint3[14937] = {X 506.0412, Y 16.5240, Z -4.6667, A 0.000, B 0.000, C 0.000 }
gfCNCPoint3[14938] = {X 506.0411, Y 40.6628, Z -4.6667, A 0.000, B 0.000, C 0.000 }
gfCNCPoint3[14939] = {X 506.6821, Y 41.4043, Z -4.6667, A 0.000, B 0.000, C 0.000 }
gfCNCPoint3[14940] = {X 507.1620, Y 42.2589, Z -4.6667, A 0.000, B 0.000, C 0.000 }
gfCNCPoint3[14941] = {X 507.4614, Y 43.1922, Z -4.6667, A 0.000, B 0.000, C 0.000 }
gfCNCPoint3[14942] = {X 507.5683, Y 44.1665, Z -4.6667, A 0.000, B 0.000, C 0.000 }
gfCNCPoint3[14943] = {X 507.5685, Y 45.0000, Z -4.6667, A 0.000, B 0.000, C 0.000 }
gfCNCPoint3[14944] = {X 507.4747, Y 45.9520, Z -4.6667, A 0.000, B 0.000, C 0.000 }
gfCNCPoint3[14945] = {X 507.1970, Y 46.8675, Z -4.6667, A 0.000, B 0.000, C 0.000 }
gfCNCPoint3[14946] = {X 506.7461, Y 47.7112, Z -4.6667, A 0.000, B 0.000, C 0.000 }
gfCNCPoint3[14947] = {X 506.1392, Y 48.4507, Z -4.6667, A 0.000, B 0.000, C 0.000 }
gfCNCPoint3[14948] = {X 505.3997, Y 49.0576, Z -4.6667, A 0.000, B 0.000, C 0.000 }
gfCNCPoint3[14949] = {X 504.5560, Y 49.5085, Z -4.6667, A 0.000, B 0.000, C 0.000 }
gfCNCPoint3[14950] = {X 503.6405, Y 49.7862, Z -4.6667, A 0.000, B 0.000, C 0.000 }
gfCNCPoint3[14951] = {X 502.6885, Y 49.8800, Z -4.6667, A 0.000, B 0.000, C 0.000 }
gfCNCPoint3[14952] = {X 496.2450, Y 49.8800, Z -4.6667, A 0.000, B 0.000, C 0.000 }
gfCNCPoint3[14953] = {X 495.2220, Y 49.7716, Z -4.6667, A 0.000, B 0.000, C 0.000 }
gfCNCPoint3[14954] = {X 494.2445, Y 49.4511, Z -4.6667, A 0.000, B 0.000, C 0.000 }
gfCNCPoint3[14955] = {X 493.3559, Y 48.9328, Z -4.6667, A 0.000, B 0.000, C 0.000 }
gfCNCPoint3[14956] = {X 492.5956, Y 48.2398, Z -4.6667, A 0.000, B 0.000, C 0.000 }
gfCNCPoint3[14957] = {X 491.9976, Y 47.4028, Z -4.6667, A 0.000, B 0.000, C 0.000 }
gfCNCPoint3[14958] = {X 491.5882, Y 46.4590, Z -4.6667, A 0.000, B 0.000, C 0.000 }
gfCNCPoint3[14959] = {X 491.4241, Y 45.7570, Z -4.6667, A 0.000, B 0.000, C 0.000 }
gfCNCPoint3[14960] = {X 491.3652, Y 45.0385, Z -4.6667, A 0.000, B 0.000, C 0.000 }
gfCNCPoint3[14961] = {X 491.3655, Y 44.1416, Z -4.6667, A 0.000, B 0.000, C 0.000 }
gfCNCPoint3[14962] = {X 491.4758, Y 43.1751, Z -4.6667, A 0.000, B 0.000, C 0.000 }
gfCNCPoint3[14963] = {X 491.7756, Y 42.2496, Z -4.6667, A 0.000, B 0.000, C 0.000 }
gfCNCPoint3[14964] = {X 492.2530, Y 41.4020, Z -4.6667, A 0.000, B 0.000, C 0.000 }
gfCNCPoint3[14965] = {X 492.8890, Y 40.6660, Z -4.6667, A 0.000, B 0.000, C 0.000 }
gfCNCPoint3[14966] = {X 492.8890, Y 35.0338, Z -4.6667, A 0.000, B 0.000, C 0.000 }
gfCNCPoint3[14967] = {X 491.0664, Y 35.0338, Z -4.6667, A 0.000, B 0.000, C 0.000 }
gfCNCPoint3[14968] = {X 487.0433, Y 42.8682, Z -4.6667, A 0.000, B 0.000, C 0.000 }
gfCNCPoint3[14969] = {X 487.1808, Y 43.5102, Z -4.6667, A 0.000, B 0.000, C 0.000 }
gfCNCPoint3[14970] = {X 487.2308, Y 44.1648, Z -4.6667, A 0.000, B 0.000, C 0.000 }
gfCNCPoint3[14971] = {X 487.2310, Y 45.0000, Z -4.6667, A 0.000, B 0.000, C 0.000 }
gfCNCPoint3[14972] = {X 487.1749, Y 45.7380, Z -4.6667, A 0.000, B 0.000, C 0.000 }
gfCNCPoint3[14973] = {X 487.0078, Y 46.4590, Z -4.6667, A 0.000, B 0.000, C 0.000 }
gfCNCPoint3[14974] = {X 486.5939, Y 47.4110, Z -4.6667, A 0.000, B 0.000, C 0.000 }
gfCNCPoint3[14975] = {X 485.9879, Y 48.2538, Z -4.6667, A 0.000, B 0.000, C 0.000 }
gfCNCPoint3[14976] = {X 485.2175, Y 48.9494, Z -4.6667, A 0.000, B 0.000, C 0.000 }
gfCNCPoint3[14977] = {X 484.3173, Y 49.4663, Z -4.6667, A 0.000, B 0.000, C 0.000 }
gfCNCPoint3[14978] = {X 483.3557, Y 49.7755, Z -4.6667, A 0.000, B 0.000, C 0.000 }
gfCNCPoint3[14979] = {X 482.3510, Y 49.8800, Z -4.6667, A 0.000, B 0.000, C 0.000 }
gfCNCPoint3[14980] = {X 480.2695, Y 49.8800, Z -4.6667, A 0.000, B 0.000, C 0.000 }
gfCNCPoint3[14981] = {X 480.2695, Y 49.4000, Z -4.6667, A 0.000, B 0.000, C 0.000 }
gfCNCPoint3[14982] = {X 475.7650, Y 49.4000, Z -4.6667, A 0.000, B 0.000, C 0.000 }
gfCNCPoint3[14983] = {X 474.7859, Y 49.2897, Z -4.6667, A 0.000, B 0.000, C 0.000 }
gfCNCPoint3[14984] = {X 473.8559, Y 48.9643, Z -4.6667, A 0.000, B 0.000, C 0.000 }
gfCNCPoint3[14985] = {X 473.0216, Y 48.4401, Z -4.6667, A 0.000, B 0.000, C 0.000 }
gfCNCPoint3[14986] = {X 472.3249, Y 47.7434, Z -4.6667, A 0.000, B 0.000, C 0.000 }
gfCNCPoint3[14987] = {X 471.8007, Y 46.9091, Z -4.6667, A 0.000, B 0.000, C 0.000 }
gfCNCPoint3[14988] = {X 471.4753, Y 45.9791, Z -4.6667, A 0.000, B 0.000, C 0.000 }
gfCNCPoint3[14989] = {X 471.3650, Y 45.0000, Z -4.6667, A 0.000, B 0.000, C 0.000 }
gfCNCPoint3[14990] = {X 471.3654, Y 44.1483, Z -4.6667, A 0.000, B 0.000, C 0.000 }
gfCNCPoint3[14991] = {X 471.4638, Y 43.2816, Z -4.6667, A 0.000, B 0.000, C 0.000 }
gfCNCPoint3[14992] = {X 471.7311, Y 42.4514, Z -4.6667, A 0.000, B 0.000, C 0.000 }
gfCNCPoint3[14993] = {X 472.1570, Y 41.6903, Z -4.6667, A 0.000, B 0.000, C 0.000 }
gfCNCPoint3[14994] = {X 472.7247, Y 41.0281, Z -4.6667, A 0.000, B 0.000, C 0.000 }
gfCNCPoint3[14995] = {X 473.4118, Y 40.4909, Z -4.6667, A 0.000, B 0.000, C 0.000 }
gfCNCPoint3[14996] = {X 474.1914, Y 40.0998, Z -4.6667, A 0.000, B 0.000, C 0.000 }
gfCNCPoint3[14997] = {X 478.1277, Y 32.3948, Z -4.6667, A 0.000, B 0.000, C 0.000 }
gfCNCPoint3[14998] = {X 476.8710, Y 31.5207, Z -4.6667, A 0.000, B 0.000, C 0.000 }
gfCNCPoint3[14999] = {X 475.7408, Y 30.4880, Z -4.6667, A 0.000, B 0.000, C 0.000 }
gfCNCPoint3[15000] = {X 474.7572, Y 29.3150, Z -4.6667, A 0.000, B 0.000, C 0.000 }
gfCNCPoint3[15001] = {X 473.9374, Y 28.0221, Z -4.6667, A 0.000, B 0.000, C 0.000 }
gfCNCPoint3[15002] = {X 473.2958, Y 26.6322, Z -4.6667, A 0.000, B 0.000, C 0.000 }
gfCNCPoint3[15003] = {X 472.8436, Y 25.1696, Z -4.6667, A 0.000, B 0.000, C 0.000 }
gfCNCPoint3[15004] = {X 472.5279, Y 23.4785, Z -4.6667, A 0.000, B 0.000, C 0.000 }
gfCNCPoint3[15005] = {X 472.3867, Y 21.7640, Z -4.6667, A 0.000, B 0.000, C 0.000 }
gfCNCPoint3[15006] = {X 472.4216, Y 20.0440, Z -4.6667, A 0.000, B 0.000, C 0.000 }
gfCNCPoint3[15007] = {X 472.6321, Y 18.3366, Z -4.6667, A 0.000, B 0.000, C 0.000 }
gfCNCPoint3[15008] = {X 473.0162, Y 16.6597, Z -4.6667, A 0.000, B 0.000, C 0.000 }
gfCNCPoint3[15009] = {X 473.5626, Y 15.1346, Z -4.6667, A 0.000, B 0.000, C 0.000 }
gfCNCPoint3[15010] = {X 474.3110, Y 13.6977, Z -4.6667, A 0.000, B 0.000, C 0.000 }
gfCNCPoint3[15011] = {X 475.2474, Y 12.3756, Z -4.6667, A 0.000, B 0.000, C 0.000 }
gfCNCPoint3[15012] = {X 476.3546, Y 11.1929, Z -4.6667, A 0.000, B 0.000, C 0.000 }
gfCNCPoint3[15013] = {X 477.6120, Y 10.1713, Z -4.6667, A 0.000, B 0.000, C 0.000 }
gfCNCPoint3[15014] = {X 478.9964, Y 9.3299, Z -4.6667, A 0.000, B 0.000, C 0.000 }
gfCNCPoint3[15015] = {X 480.4822, Y 8.6840, Z -4.6667, A 0.000, B 0.000, C 0.000 }
gfCNCPoint3[15016] = {X 482.0419, Y 8.2458, Z -4.6667, A 0.000, B 0.000, C 0.000 }
gfCNCPoint3[15017] = {X 484.1468, Y 7.9178, Z -4.6667, A 0.000, B 0.000, C 0.000 }
gfCNCPoint3[15018] = {X 486.2739, Y 7.8027, Z -4.6667, A 0.000, B 0.000, C 0.000 }
gfCNCPoint3[15019] = {X 486.9707, Y 7.7906, Z -4.6667, A 0.000, B 0.000, C 0.000 }
gfCNCPoint3[15020] = {X 502.2084, Y 7.7906, Z -4.6667, A 0.000, B 0.000, C 0.000 }
gfCNCPoint3[15021] = {X 502.7401, Y 7.7947, Z -4.6667, A 0.000, B 0.000, C 0.000 }
gfCNCPoint3[15022] = {X 503.7096, Y 7.9111, Z -4.6667, A 0.000, B 0.000, C 0.000 }
gfCNCPoint3[15023] = {X 504.6294, Y 8.2393, Z -4.6667, A 0.000, B 0.000, C 0.000 }
gfCNCPoint3[15024] = {X 505.4536, Y 8.7630, Z -4.6667, A 0.000, B 0.000, C 0.000 }
gfCNCPoint3[15025] = {X 506.1415, Y 9.4562, Z -4.6667, A 0.000, B 0.000, C 0.000 }
gfCNCPoint3[15026] = {X 506.6587, Y 10.2845, Z -4.6667, A 0.000, B 0.000, C 0.000 }
gfCNCPoint3[15027] = {X 506.9797, Y 11.2068, Z -4.6667, A 0.000, B 0.000, C 0.000 }
gfCNCPoint3[15028] = {X 507.0885, Y 12.1773, Z -4.6667, A 0.000, B 0.000, C 0.000 }
gfCNCPoint3[15029] = {X 507.0883, Y 13.0233, Z -4.6667, A 0.000, B 0.000, C 0.000 }
gfCNCPoint3[15030] = {X 506.9800, Y 13.9493, Z -4.6667, A 0.000, B 0.000, C 0.000 }
gfCNCPoint3[15031] = {X 506.6790, Y 14.8316, Z -4.6667, A 0.000, B 0.000, C 0.000 }
gfCNCPoint3[15032] = {X 506.1989, Y 15.6308, Z -4.6667, A 0.000, B 0.000, C 0.000 }
gfCNCPoint3[15033] = {X 505.5612, Y 16.3108, Z -4.6667, A 0.000, B 0.000, C 0.000 }
gfCNCPoint3[15034] = {X 505.5611, Y 40.8759, Z -4.6667, A 0.000, B 0.000, C 0.000 }
gfCNCPoint3[15035] = {X 506.2057, Y 41.5651, Z -4.6667, A 0.000, B 0.000, C 0.000 }
gfCNCPoint3[15036] = {X 506.6885, Y 42.3758, Z -4.6667, A 0.000, B 0.000, C 0.000 }
gfCNCPoint3[15037] = {X 506.9873, Y 43.2708, Z -4.6667, A 0.000, B 0.000, C 0.000 }
gfCNCPoint3[15038] = {X 507.0885, Y 44.2089, Z -4.6667, A 0.000, B 0.000, C 0.000 }
gfCNCPoint3[15039] = {X 507.0885, Y 45.0000, Z -4.6667, A 0.000, B 0.000, C 0.000 }
gfCNCPoint3[15040] = {X 506.9782, Y 45.9791, Z -4.6667, A 0.000, B 0.000, C 0.000 }
gfCNCPoint3[15041] = {X 506.6528, Y 46.9091, Z -4.6667, A 0.000, B 0.000, C 0.000 }
gfCNCPoint3[15042] = {X 506.1285, Y 47.7434, Z -4.6667, A 0.000, B 0.000, C 0.000 }
gfCNCPoint3[15043] = {X 505.4318, Y 48.4401, Z -4.6667, A 0.000, B 0.000, C 0.000 }
gfCNCPoint3[15044] = {X 504.5976, Y 48.9643, Z -4.6667, A 0.000, B 0.000, C 0.000 }
gfCNCPoint3[15045] = {X 503.6676, Y 49.2897, Z -4.6667, A 0.000, B 0.000, C 0.000 }
gfCNCPoint3[15046] = {X 502.6885, Y 49.4000, Z -4.6667, A 0.000, B 0.000, C 0.000 }
gfCNCPoint3[15047] = {X 496.2450, Y 49.4000, Z -4.6667, A 0.000, B 0.000, C 0.000 }
gfCNCPoint3[15048] = {X 495.2659, Y 49.2897, Z -4.6667, A 0.000, B 0.000, C 0.000 }
gfCNCPoint3[15049] = {X 494.3359, Y 48.9643, Z -4.6667, A 0.000, B 0.000, C 0.000 }
gfCNCPoint3[15050] = {X 493.5017, Y 48.4400, Z -4.6667, A 0.000, B 0.000, C 0.000 }
gfCNCPoint3[15051] = {X 492.8050, Y 47.7433, Z -4.6667, A 0.000, B 0.000, C 0.000 }
gfCNCPoint3[15052] = {X 492.2808, Y 46.9091, Z -4.6667, A 0.000, B 0.000, C 0.000 }
gfCNCPoint3[15053] = {X 491.9553, Y 45.9791, Z -4.6667, A 0.000, B 0.000, C 0.000 }
gfCNCPoint3[15054] = {X 491.8450, Y 45.0000, Z -4.6667, A 0.000, B 0.000, C 0.000 }
gfCNCPoint3[15055] = {X 491.8454, Y 44.1483, Z -4.6667, A 0.000, B 0.000, C 0.000 }
gfCNCPoint3[15056] = {X 491.9559, Y 43.2275, Z -4.6667, A 0.000, B 0.000, C 0.000 }
gfCNCPoint3[15057] = {X 492.2568, Y 42.3503, Z -4.6667, A 0.000, B 0.000, C 0.000 }
gfCNCPoint3[15058] = {X 492.7349, Y 41.5556, Z -4.6667, A 0.000, B 0.000, C 0.000 }
gfCNCPoint3[15059] = {X 493.3690, Y 40.8789, Z -4.6667, A 0.000, B 0.000, C 0.000 }
gfCNCPoint3[15060] = {X 493.3690, Y 34.5538, Z -4.6667, A 0.000, B 0.000, C 0.000 }
gfCNCPoint3[15061] = {X 490.7733, Y 34.5538, Z -4.6667, A 0.000, B 0.000, C 0.000 }
gfCNCPoint3[15062] = {X 486.5270, Y 42.8228, Z -4.6667, A 0.000, B 0.000, C 0.000 }
gfCNCPoint3[15063] = {X 486.6947, Y 43.5068, Z -4.6667, A 0.000, B 0.000, C 0.000 }
gfCNCPoint3[15064] = {X 486.7510, Y 44.2089, Z -4.6667, A 0.000, B 0.000, C 0.000 }
gfCNCPoint3[15065] = {X 486.7510, Y 45.0000, Z -4.6667, A 0.000, B 0.000, C 0.000 }
gfCNCPoint3[15066] = {X 486.6407, Y 45.9791, Z -4.6667, A 0.000, B 0.000, C 0.000 }
gfCNCPoint3[15067] = {X 486.3153, Y 46.9091, Z -4.6667, A 0.000, B 0.000, C 0.000 }
gfCNCPoint3[15068] = {X 485.7911, Y 47.7434, Z -4.6667, A 0.000, B 0.000, C 0.000 }
gfCNCPoint3[15069] = {X 485.0944, Y 48.4401, Z -4.6667, A 0.000, B 0.000, C 0.000 }
gfCNCPoint3[15070] = {X 484.2601, Y 48.9643, Z -4.6667, A 0.000, B 0.000, C 0.000 }
gfCNCPoint3[15071] = {X 483.3301, Y 49.2897, Z -4.6667, A 0.000, B 0.000, C 0.000 }
gfCNCPoint3[15072] = {X 482.3510, Y 49.4000, Z -4.6667, A 0.000, B 0.000, C 0.000 }
gfCNCPoint3[15073] = {X 480.2695, Y 49.4000, Z -4.6667, A 0.000, B 0.000, C 0.000 }
gfCNCPoint3[15074] = {X 480.2695, Y 49.8800, Z -4.6667, A 0.000, B 0.000, C 0.000 }
gfCNCPoint3[15075] = {X 481.4067, Y 50.7435, Z -4.6667, A 0.000, B 0.000, C 0.000 }
gfCNCPoint3[15076] = {X 482.4044, Y 51.7649, Z -4.6667, A 0.000, B 0.000, C 0.000 }
gfCNCPoint3[15077] = {X 483.2411, Y 52.9219, Z -4.6667, A 0.000, B 0.000, C 0.000 }
gfCNCPoint3[15078] = {X 483.8615, Y 54.1044, Z -4.6667, A 0.000, B 0.000, C 0.000 }
gfCNCPoint3[15079] = {X 484.3133, Y 55.3610, Z -4.6667, A 0.000, B 0.000, C 0.000 }
gfCNCPoint3[15080] = {X 484.5879, Y 56.6678, Z -4.6667, A 0.000, B 0.000, C 0.000 }
gfCNCPoint3[15081] = {X 484.6800, Y 58.0000, Z -4.6667, A 0.000, B 0.000, C 0.000 }
gfCNCPoint3[15082] = {X 484.6797, Y 59.0140, Z -4.6667, A 0.000, B 0.000, C 0.000 }
gfCNCPoint3[15083] = {X 484.5592, Y 60.4584, Z -4.6667, A 0.000, B 0.000, C 0.000 }
gfCNCPoint3[15084] = {X 484.2245, Y 61.8686, Z -4.6667, A 0.000, B 0.000, C 0.000 }
gfCNCPoint3[15085] = {X 483.6829, Y 63.2130, Z -4.6667, A 0.000, B 0.000, C 0.000 }
gfCNCPoint3[15086] = {X 482.9467, Y 64.4615, Z -4.6667, A 0.000, B 0.000, C 0.000 }
gfCNCPoint3[15087] = {X 482.0323, Y 65.5861, Z -4.6667, A 0.000, B 0.000, C 0.000 }
gfCNCPoint3[15088] = {X 480.9603, Y 66.5615, Z -4.6667, A 0.000, B 0.000, C 0.000 }
gfCNCPoint3[15089] = {X 480.9606, Y 89.4443, Z -4.6667, A 0.000, B 0.000, C 0.000 }
gfCNCPoint3[15090] = {X 482.0603, Y 90.4466, Z -4.6667, A 0.000, B 0.000, C 0.000 }
gfCNCPoint3[15091] = {X 482.9928, Y 91.6061, Z -4.6667, A 0.000, B 0.000, C 0.000 }
gfCNCPoint3[15092] = {X 483.7361, Y 92.8950, Z -4.6667, A 0.000, B 0.000, C 0.000 }
gfCNCPoint3[15093] = {X 507.6815, Y 92.8950, Z -4.6667, A 0.000, B 0.000, C 0.000 }
gfCNCPoint3[15094] = {X 507.6815, Y 95.2950, Z -4.6667, A 0.000, B 0.000, C 0.000 }
gfCNCPoint3[15095] = {X 595.2966, Y 95.2950, Z -4.6667, A 0.000, B 0.000, C 0.000 }
gfCNCPoint3[15096] = {X 595.2966, Y 54.2000, Z -4.6667, A 0.000, B 0.000, C 0.000 }
gfCNCPoint3[15097] = {X 593.5565, Y 54.2000, Z -4.6667, A 0.000, B 0.000, C 0.000 }
gfCNCPoint3[15098] = {X 592.2403, Y 54.1053, Z -4.6667, A 0.000, B 0.000, C 0.000 }
gfCNCPoint3[15099] = {X 590.9511, Y 53.8233, Z -4.6667, A 0.000, B 0.000, C 0.000 }
gfCNCPoint3[15100] = {X 589.7155, Y 53.3598, Z -4.6667, A 0.000, B 0.000, C 0.000 }
gfCNCPoint3[15101] = {X 588.5589, Y 52.7242, Z -4.6667, A 0.000, B 0.000, C 0.000 }
gfCNCPoint3[15102] = {X 587.5052, Y 51.9297, Z -4.6667, A 0.000, B 0.000, C 0.000 }
gfCNCPoint3[15103] = {X 586.4956, Y 52.6955, Z -4.6667, A 0.000, B 0.000, C 0.000 }
gfCNCPoint3[15104] = {X 585.3903, Y 53.3153, Z -4.6667, A 0.000, B 0.000, C 0.000 }
gfCNCPoint3[15105] = {X 584.1375, Y 53.7999, Z -4.6667, A 0.000, B 0.000, C 0.000 }
gfCNCPoint3[15106] = {X 582.8276, Y 54.0969, Z -4.6667, A 0.000, B 0.000, C 0.000 }
gfCNCPoint3[15107] = {X 581.4884, Y 54.1999, Z -4.6667, A 0.000, B 0.000, C 0.000 }
gfCNCPoint3[15108] = {X 580.1485, Y 54.1069, Z -4.6667, A 0.000, B 0.000, C 0.000 }
gfCNCPoint3[15109] = {X 578.8364, Y 53.8198, Z -4.6667, A 0.000, B 0.000, C 0.000 }
gfCNCPoint3[15110] = {X 577.5801, Y 53.3447, Z -4.6667, A 0.000, B 0.000, C 0.000 }
gfCNCPoint3[15111] = {X 576.4063, Y 52.6917, Z -4.6667, A 0.000, B 0.000, C 0.000 }
gfCNCPoint3[15112] = {X 575.3401, Y 51.8748, Z -4.6667, A 0.000, B 0.000, C 0.000 }
gfCNCPoint3[15113] = {X 574.2798, Y 52.6879, Z -4.6667, A 0.000, B 0.000, C 0.000 }
gfCNCPoint3[15114] = {X 573.1128, Y 53.3388, Z -4.6667, A 0.000, B 0.000, C 0.000 }
gfCNCPoint3[15115] = {X 571.8638, Y 53.8139, Z -4.6667, A 0.000, B 0.000, C 0.000 }
gfCNCPoint3[15116] = {X 570.5592, Y 54.1030, Z -4.6667, A 0.000, B 0.000, C 0.000 }
gfCNCPoint3[15117] = {X 569.2264, Y 54.2000, Z -4.6667, A 0.000, B 0.000, C 0.000 }
gfCNCPoint3[15118] = {X 562.4443, Y 54.2000, Z -4.6667, A 0.000, B 0.000, C 0.000 }
gfCNCPoint3[15119] = {X 561.0051, Y 54.0867, Z -4.6667, A 0.000, B 0.000, C 0.000 }
gfCNCPoint3[15120] = {X 559.6013, Y 53.7497, Z -4.6667, A 0.000, B 0.000, C 0.000 }
gfCNCPoint3[15121] = {X 558.2676, Y 53.1973, Z -4.6667, A 0.000, B 0.000, C 0.000 }
gfCNCPoint3[15122] = {X 557.0367, Y 52.4430, Z -4.6667, A 0.000, B 0.000, C 0.000 }
gfCNCPoint3[15123] = {X 555.9389, Y 51.5054, Z -4.6667, A 0.000, B 0.000, C 0.000 }
gfCNCPoint3[15124] = {X 555.0013, Y 50.4076, Z -4.6667, A 0.000, B 0.000, C 0.000 }
gfCNCPoint3[15125] = {X 554.2470, Y 49.1767, Z -4.6667, A 0.000, B 0.000, C 0.000 }
gfCNCPoint3[15126] = {X 553.6946, Y 47.8430, Z -4.6667, A 0.000, B 0.000, C 0.000 }
gfCNCPoint3[15127] = {X 553.3576, Y 46.4392, Z -4.6667, A 0.000, B 0.000, C 0.000 }
gfCNCPoint3[15128] = {X 553.2443, Y 45.0000, Z -4.6667, A 0.000, B 0.000, C 0.000 }
gfCNCPoint3[15129] = {X 553.2443, Y 44.0446, Z -4.6667, A 0.000, B 0.000, C 0.000 }
gfCNCPoint3[15130] = {X 553.3465, Y 42.7123, Z -4.6667, A 0.000, B 0.000, C 0.000 }
gfCNCPoint3[15131] = {X 553.6399, Y 41.4088, Z -4.6667, A 0.000, B 0.000, C 0.000 }
gfCNCPoint3[15132] = {X 554.1183, Y 40.1612, Z -4.6667, A 0.000, B 0.000, C 0.000 }
gfCNCPoint3[15133] = {X 554.7718, Y 38.9957, Z -4.6667, A 0.000, B 0.000, C 0.000 }
gfCNCPoint3[15134] = {X 554.7718, Y 11.0107, Z -4.6667, A 0.000, B 0.000, C 0.000 }
gfCNCPoint3[15135] = {X 554.1219, Y 9.8554, Z -4.6667, A 0.000, B 0.000, C 0.000 }
gfCNCPoint3[15136] = {X 553.6447, Y 8.6188, Z -4.6667, A 0.000, B 0.000, C 0.000 }
gfCNCPoint3[15137] = {X 553.3503, Y 7.3264, Z -4.6667, A 0.000, B 0.000, C 0.000 }
gfCNCPoint3[15138] = {X 553.2446, Y 6.0051, Z -4.6667, A 0.000, B 0.000, C 0.000 }
gfCNCPoint3[15139] = {X 553.2443, Y 5.0000, Z -4.6667, A 0.000, B 0.000, C 0.000 }
gfCNCPoint3[15140] = {X 553.2455, Y 4.8525, Z -4.6667, A 0.000, B 0.000, C 0.000 }
gfCNCPoint3[15141] = {X 553.2490, Y 4.7050, Z -4.6667, A 0.000, B 0.000, C 0.000 }
gfCNCPoint3[15142] = {X 365.1872, Y 4.7050, Z -4.6667, A 0.000, B 0.000, C 0.000 }
gfCNCPoint3[15143] = {X 365.5720, Y 5.1238, Z -4.6667, A 0.000, B 0.000, C 0.000 }
gfCNCPoint3[15144] = {X 365.9468, Y 5.5516, Z -4.6667, A 0.000, B 0.000, C 0.000 }
gfCNCPoint3[15145] = {X 367.0661, Y 6.9493, Z -4.6667, A 0.000, B 0.000, C 0.000 }
gfCNCPoint3[15146] = {X 368.0928, Y 8.4166, Z -4.6667, A 0.000, B 0.000, C 0.000 }
gfCNCPoint3[15147] = {X 369.3403, Y 10.5271, Z -4.6667, A 0.000, B 0.000, C 0.000 }
gfCNCPoint3[15148] = {X 370.3963, Y 12.7397, Z -4.6667, A 0.000, B 0.000, C 0.000 }
gfCNCPoint3[15149] = {X 371.2522, Y 15.0371, Z -4.6667, A 0.000, B 0.000, C 0.000 }
gfCNCPoint3[15150] = {X 371.9015, Y 17.4012, Z -4.6667, A 0.000, B 0.000, C 0.000 }
gfCNCPoint3[15151] = {X 372.3592, Y 19.8024, Z -4.6667, A 0.000, B 0.000, C 0.000 }
gfCNCPoint3[15152] = {X 372.6462, Y 22.2299, Z -4.6667, A 0.000, B 0.000, C 0.000 }
gfCNCPoint3[15153] = {X 372.7608, Y 24.6717, Z -4.6667, A 0.000, B 0.000, C 0.000 }
gfCNCPoint3[15154] = {X 372.7026, Y 27.1154, Z -4.6667, A 0.000, B 0.000, C 0.000 }
gfCNCPoint3[15155] = {X 372.4719, Y 29.5490, Z -4.6667, A 0.000, B 0.000, C 0.000 }
gfCNCPoint3[15156] = {X 372.0698, Y 31.9601, Z -4.6667, A 0.000, B 0.000, C 0.000 }
gfCNCPoint3[15157] = {X 371.4836, Y 34.3146, Z -4.6667, A 0.000, B 0.000, C 0.000 }
gfCNCPoint3[15158] = {X 370.6920, Y 36.6082, Z -4.6667, A 0.000, B 0.000, C 0.000 }
gfCNCPoint3[15159] = {X 369.7013, Y 38.8231, Z -4.6667, A 0.000, B 0.000, C 0.000 }
gfCNCPoint3[15160] = {X 368.5190, Y 40.9420, Z -4.6667, A 0.000, B 0.000, C 0.000 }
gfCNCPoint3[15161] = {X 367.1545, Y 42.9483, Z -4.6667, A 0.000, B 0.000, C 0.000 }
gfCNCPoint3[15162] = {X 367.0319, Y 43.1164, Z -4.6667, A 0.000, B 0.000, C 0.000 }
gfCNCPoint3[15163] = {X 366.9644, Y 43.2038, Z -4.6667, A 0.000, B 0.000, C 0.000 }
gfCNCPoint3[15164] = {X 366.3199, Y 43.9953, Z -4.6667, A 0.000, B 0.000, C 0.000 }
gfCNCPoint3[15165] = {X 364.8835, Y 45.6070, Z -4.6667, A 0.000, B 0.000, C 0.000 }
gfCNCPoint3[15166] = {X 363.3095, Y 47.0845, Z -4.6667, A 0.000, B 0.000, C 0.000 }
gfCNCPoint3[15167] = {X 361.6104, Y 48.4163, Z -4.6667, A 0.000, B 0.000, C 0.000 }
gfCNCPoint3[15168] = {X 359.7996, Y 49.5918, Z -4.6667, A 0.000, B 0.000, C 0.000 }
gfCNCPoint3[15169] = {X 357.8915, Y 50.6016, Z -4.6667, A 0.000, B 0.000, C 0.000 }
gfCNCPoint3[15170] = {X 357.4231, Y 50.8220, Z -4.6667, A 0.000, B 0.000, C 0.000 }
gfCNCPoint3[15171] = {X 355.4490, Y 51.5846, Z -4.6667, A 0.000, B 0.000, C 0.000 }
gfCNCPoint3[15172] = {X 353.4194, Y 52.1840, Z -4.6667, A 0.000, B 0.000, C 0.000 }
gfCNCPoint3[15173] = {X 351.3477, Y 52.6162, Z -4.6667, A 0.000, B 0.000, C 0.000 }
gfCNCPoint3[15174] = {X 349.2477, Y 52.8784, Z -4.6667, A 0.000, B 0.000, C 0.000 }
gfCNCPoint3[15175] = {X 347.1334, Y 52.9689, Z -4.6667, A 0.000, B 0.000, C 0.000 }
gfCNCPoint3[15176] = {X 344.8132, Y 52.9266, Z -4.6667, A 0.000, B 0.000, C 0.000 }
gfCNCPoint3[15177] = {X 342.5053, Y 52.6835, Z -4.6667, A 0.000, B 0.000, C 0.000 }
gfCNCPoint3[15178] = {X 340.2272, Y 52.2414, Z -4.6667, A 0.000, B 0.000, C 0.000 }
gfCNCPoint3[15179] = {X 337.9959, Y 51.6036, Z -4.6667, A 0.000, B 0.000, C 0.000 }
gfCNCPoint3[15180] = {X 335.8283, Y 50.7750, Z -4.6667, A 0.000, B 0.000, C 0.000 }
gfCNCPoint3[15181] = {X 333.7406, Y 49.7618, Z -4.6667, A 0.000, B 0.000, C 0.000 }
gfCNCPoint3[15182] = {X 332.8357, Y 49.2292, Z -4.6667, A 0.000, B 0.000, C 0.000 }
gfCNCPoint3[15183] = {X 331.9523, Y 48.6616, Z -4.6667, A 0.000, B 0.000, C 0.000 }
gfCNCPoint3[15184] = {X 331.3028, Y 48.2120, Z -4.6667, A 0.000, B 0.000, C 0.000 }
gfCNCPoint3[15185] = {X 330.6669, Y 47.7434, Z -4.6667, A 0.000, B 0.000, C 0.000 }
gfCNCPoint3[15186] = {X 329.2148, Y 49.6542, Z -4.6667, A 0.000, B 0.000, C 0.000 }
gfCNCPoint3[15187] = {X 328.8710, Y 49.3889, Z -4.6667, A 0.000, B 0.000, C 0.000 }
gfCNCPoint3[15188] = {X 328.5312, Y 49.1185, Z -4.6667, A 0.000, B 0.000, C 0.000 }
gfCNCPoint3[15189] = {X 328.1264, Y 49.0390, Z -4.6667, A 0.000, B 0.000, C 0.000 }
gfCNCPoint3[15190] = {X 327.7253, Y 48.9423, Z -4.6667, A 0.000, B 0.000, C 0.000 }
gfCNCPoint3[15191] = {X 328.4853, Y 49.2664, Z -4.6667, A 0.000, B 0.000, C 0.000 }
gfCNCPoint3[15192] = {X 329.2148, Y 49.6542, Z -4.6667, A 0.000, B 0.000, C 0.000 }
gfCNCPoint3[15193] = {X 330.6669, Y 47.7434, Z -4.6667, A 0.000, B 0.000, C 0.000 }
gfCNCPoint3[15194] = {X 330.0940, Y 47.2956, Z -4.6667, A 0.000, B 0.000, C 0.000 }
gfCNCPoint3[15195] = {X 329.5334, Y 46.8324, Z -4.6667, A 0.000, B 0.000, C 0.000 }
gfCNCPoint3[15196] = {X 328.9310, Y 46.7520, Z -4.6667, A 0.000, B 0.000, C 0.000 }
gfCNCPoint3[15197] = {X 328.3374, Y 46.6216, Z -4.6667, A 0.000, B 0.000, C 0.000 }
gfCNCPoint3[15198] = {X 327.9789, Y 46.5172, Z -4.6667, A 0.000, B 0.000, C 0.000 }
gfCNCPoint3[15199] = {X 327.6263, Y 46.3944, Z -4.6667, A 0.000, B 0.000, C 0.000 }
gfCNCPoint3[15200] = {X 326.7320, Y 45.9864, Z -4.6667, A 0.000, B 0.000, C 0.000 }
gfCNCPoint3[15201] = {X 325.9009, Y 45.4616, Z -4.6667, A 0.000, B 0.000, C 0.000 }
gfCNCPoint3[15202] = {X 325.1480, Y 44.8296, Z -4.6667, A 0.000, B 0.000, C 0.000 }
gfCNCPoint3[15203] = {X 324.5140, Y 44.2115, Z -4.6667, A 0.000, B 0.000, C 0.000 }
gfCNCPoint3[15204] = {X 324.0475, Y 43.7117, Z -4.6667, A 0.000, B 0.000, C 0.000 }
gfCNCPoint3[15205] = {X 323.6300, Y 43.1703, Z -4.6667, A 0.000, B 0.000, C 0.000 }
gfCNCPoint3[15206] = {X 319.6957, Y 45.9200, Z -4.6667, A 0.000, B 0.000, C 0.000 }
gfCNCPoint3[15207] = {X 319.4780, Y 45.5976, Z -4.6667, A 0.000, B 0.000, C 0.000 }
gfCNCPoint3[15208] = {X 319.2708, Y 45.2683, Z -4.6667, A 0.000, B 0.000, C 0.000 }
gfCNCPoint3[15209] = {X 319.2514, Y 45.5948, Z -4.6667, A 0.000, B 0.000, C 0.000 }
gfCNCPoint3[15210] = {X 319.2174, Y 45.9200, Z -4.6667, A 0.000, B 0.000, C 0.000 }
gfCNCPoint3[15211] = {X 319.6957, Y 45.9200, Z -4.6667, A 0.000, B 0.000, C 0.000 }
gfCNCPoint3[15212] = {X 321.6628, Y 44.5452, Z -4.6667, A 0.000, B 0.000, C 0.000 }
gfCNCPoint3[15213] = {X 321.4884, Y 44.2868, Z -4.6667, A 0.000, B 0.000, C 0.000 }
gfCNCPoint3[15214] = {X 321.3224, Y 44.0230, Z -4.6667, A 0.000, B 0.000, C 0.000 }
gfCNCPoint3[15215] = {X 320.6710, Y 42.7451, Z -4.6667, A 0.000, B 0.000, C 0.000 }
gfCNCPoint3[15216] = {X 320.2156, Y 41.3851, Z -4.6667, A 0.000, B 0.000, C 0.000 }
gfCNCPoint3[15217] = {X 319.9662, Y 39.9727, Z -4.6667, A 0.000, B 0.000, C 0.000 }
gfCNCPoint3[15218] = {X 319.9282, Y 38.5389, Z -4.6667, A 0.000, B 0.000, C 0.000 }
gfCNCPoint3[15219] = {X 320.1024, Y 37.1153, Z -4.6667, A 0.000, B 0.000, C 0.000 }
gfCNCPoint3[15220] = {X 320.4305, Y 35.8896, Z -4.6667, A 0.000, B 0.000, C 0.000 }
gfCNCPoint3[15221] = {X 320.9161, Y 34.7173, Z -4.6667, A 0.000, B 0.000, C 0.000 }
gfCNCPoint3[15222] = {X 321.5508, Y 33.6186, Z -4.6667, A 0.000, B 0.000, C 0.000 }
gfCNCPoint3[15223] = {X 324.1388, Y 29.7491, Z -4.6667, A 0.000, B 0.000, C 0.000 }
gfCNCPoint3[15224] = {X 320.1489, Y 27.0806, Z -4.6667, A 0.000, B 0.000, C 0.000 }
gfCNCPoint3[15225] = {X 321.8043, Y 24.6055, Z -4.6667, A 0.000, B 0.000, C 0.000 }
gfCNCPoint3[15226] = {X 321.9898, Y 24.3355, Z -4.6667, A 0.000, B 0.000, C 0.000 }
gfCNCPoint3[15227] = {X 322.1814, Y 24.0697, Z -4.6667, A 0.000, B 0.000, C 0.000 }
gfCNCPoint3[15228] = {X 321.5380, Y 23.0772, Z -4.6667, A 0.000, B 0.000, C 0.000 }
gfCNCPoint3[15229] = {X 320.9777, Y 22.0354, Z -4.6667, A 0.000, B 0.000, C 0.000 }
gfCNCPoint3[15230] = {X 320.1493, Y 20.3313, Z -4.6667, A 0.000, B 0.000, C 0.000 }
gfCNCPoint3[15231] = {X 320.1489, Y 27.0806, Z -4.6667, A 0.000, B 0.000, C 0.000 }
gfCNCPoint3[15232] = {X 322.1439, Y 28.4149, Z -4.6667, A 0.000, B 0.000, C 0.000 }
gfCNCPoint3[15233] = {X 323.7976, Y 25.9422, Z -4.6667, A 0.000, B 0.000, C 0.000 }
gfCNCPoint3[15234] = {X 324.5113, Y 24.9840, Z -4.6667, A 0.000, B 0.000, C 0.000 }
gfCNCPoint3[15235] = {X 325.3162, Y 24.1010, Z -4.6667, A 0.000, B 0.000, C 0.000 }
gfCNCPoint3[15236] = {X 324.4812, Y 23.1413, Z -4.6667, A 0.000, B 0.000, C 0.000 }
gfCNCPoint3[15237] = {X 323.7518, Y 22.0991, Z -4.6667, A 0.000, B 0.000, C 0.000 }
gfCNCPoint3[15238] = {X 323.1360, Y 20.9859, Z -4.6667, A 0.000, B 0.000, C 0.000 }
gfCNCPoint3[15239] = {X 319.6151, Y 13.7428, Z -4.6667, A 0.000, B 0.000, C 0.000 }
gfCNCPoint3[15240] = {X 319.4387, Y 13.3633, Z -4.6667, A 0.000, B 0.000, C 0.000 }
gfCNCPoint3[15241] = {X 319.2755, Y 12.9779, Z -4.6667, A 0.000, B 0.000, C 0.000 }
gfCNCPoint3[15242] = {X 319.2755, Y 13.0353, Z -4.6667, A 0.000, B 0.000, C 0.000 }
gfCNCPoint3[15243] = {X 319.1698, Y 14.2151, Z -4.6667, A 0.000, B 0.000, C 0.000 }
gfCNCPoint3[15244] = {X 318.8743, Y 15.3621, Z -4.6667, A 0.000, B 0.000, C 0.000 }
gfCNCPoint3[15245] = {X 318.3966, Y 16.4461, Z -4.6667, A 0.000, B 0.000, C 0.000 }
gfCNCPoint3[15246] = {X 317.7495, Y 17.4382, Z -4.6667, A 0.000, B 0.000, C 0.000 }
gfCNCPoint3[15247] = {X 317.7483, Y 36.6480, Z -4.6667, A 0.000, B 0.000, C 0.000 }
gfCNCPoint3[15248] = {X 318.1578, Y 35.1184, Z -4.6667, A 0.000, B 0.000, C 0.000 }
gfCNCPoint3[15249] = {X 318.7638, Y 33.6555, Z -4.6667, A 0.000, B 0.000, C 0.000 }
gfCNCPoint3[15250] = {X 319.5559, Y 32.2844, Z -4.6667, A 0.000, B 0.000, C 0.000 }
gfCNCPoint3[15251] = {X 322.1439, Y 28.4149, Z -4.6667, A 0.000, B 0.000, C 0.000 }
gfCNCPoint3[15252] = {X 324.1388, Y 29.7491, Z -4.6667, A 0.000, B 0.000, C 0.000 }
gfCNCPoint3[15253] = {X 325.7909, Y 27.2789, Z -4.6667, A 0.000, B 0.000, C 0.000 }
gfCNCPoint3[15254] = {X 326.3628, Y 26.5111, Z -4.6667, A 0.000, B 0.000, C 0.000 }
gfCNCPoint3[15255] = {X 327.0077, Y 25.8035, Z -4.6667, A 0.000, B 0.000, C 0.000 }
gfCNCPoint3[15256] = {X 328.0707, Y 24.8904, Z -4.6667, A 0.000, B 0.000, C 0.000 }
gfCNCPoint3[15257] = {X 329.2543, Y 24.1403, Z -4.6667, A 0.000, B 0.000, C 0.000 }
gfCNCPoint3[15258] = {X 328.0859, Y 23.3667, Z -4.6667, A 0.000, B 0.000, C 0.000 }
gfCNCPoint3[15259] = {X 327.0414, Y 22.4326, Z -4.6667, A 0.000, B 0.000, C 0.000 }
gfCNCPoint3[15260] = {X 326.3723, Y 21.6635, Z -4.6667, A 0.000, B 0.000, C 0.000 }
gfCNCPoint3[15261] = {X 325.7878, Y 20.8284, Z -4.6667, A 0.000, B 0.000, C 0.000 }
gfCNCPoint3[15262] = {X 325.2944, Y 19.9364, Z -4.6667, A 0.000, B 0.000, C 0.000 }
gfCNCPoint3[15263] = {X 321.7736, Y 12.6936, Z -4.6667, A 0.000, B 0.000, C 0.000 }
gfCNCPoint3[15264] = {X 321.6322, Y 12.3894, Z -4.6667, A 0.000, B 0.000, C 0.000 }
gfCNCPoint3[15265] = {X 321.5015, Y 12.0806, Z -4.6667, A 0.000, B 0.000, C 0.000 }
gfCNCPoint3[15266] = {X 321.1058, Y 10.8774, Z -4.6667, A 0.000, B 0.000, C 0.000 }
gfCNCPoint3[15267] = {X 320.8706, Y 9.6327, Z -4.6667, A 0.000, B 0.000, C 0.000 }
gfCNCPoint3[15268] = {X 320.7999, Y 8.3681, Z -4.6667, A 0.000, B 0.000, C 0.000 }
gfCNCPoint3[15269] = {X 320.8950, Y 7.1050, Z -4.6667, A 0.000, B 0.000, C 0.000 }
gfCNCPoint3[15270] = {X 298.7842, Y 7.1050, Z -4.6667, A 0.000, B 0.000, C 0.000 }
gfCNCPoint3[15271] = {X 298.7842, Y 9.5050, Z -4.6667, A 0.000, B 0.000, C 0.000 }
gfCNCPoint3[15272] = {X 297.8292, Y 9.5050, Z -4.6667, A 0.000, B 0.000, C 0.000 }
gfCNCPoint3[15273] = {X 298.1371, Y 10.4755, Z -4.6667, A 0.000, B 0.000, C 0.000 }
gfCNCPoint3[15274] = {X 298.3067, Y 11.4795, Z -4.6667, A 0.000, B 0.000, C 0.000 }
gfCNCPoint3[15275] = {X 298.4763, Y 10.4755, Z -4.6667, A 0.000, B 0.000, C 0.000 }
gfCNCPoint3[15276] = {X 298.7842, Y 9.5050, Z -4.6667, A 0.000, B 0.000, C 0.000 }
gfCNCPoint3[15277] = {X 298.7842, Y 7.1050, Z -4.6667, A 0.000, B 0.000, C 0.000 }
gfCNCPoint3[15278] = {X 233.3044, Y 7.1050, Z -4.6667, A 0.000, B 0.000, C 0.000 }
gfCNCPoint3[15279] = {X 233.3044, Y 11.9050, Z -4.6667, A 0.000, B 0.000, C 0.000 }
gfCNCPoint3[15280] = {X 233.1564, Y 11.9050, Z -4.6667, A 0.000, B 0.000, C 0.000 }
gfCNCPoint3[15281] = {X 233.1594, Y 12.0448, Z -4.6667, A 0.000, B 0.000, C 0.000 }
gfCNCPoint3[15282] = {X 233.1605, Y 12.1847, Z -4.6667, A 0.000, B 0.000, C 0.000 }
gfCNCPoint3[15283] = {X 233.2318, Y 12.0445, Z -4.6667, A 0.000, B 0.000, C 0.000 }
gfCNCPoint3[15284] = {X 233.3044, Y 11.9050, Z -4.6667, A 0.000, B 0.000, C 0.000 }
gfCNCPoint3[15285] = {X 233.3044, Y 9.5050, Z -4.6667, A 0.000, B 0.000, C 0.000 }
gfCNCPoint3[15286] = {X 230.2485, Y 9.5050, Z -4.6667, A 0.000, B 0.000, C 0.000 }
gfCNCPoint3[15287] = {X 230.6107, Y 10.7177, Z -4.6667, A 0.000, B 0.000, C 0.000 }
gfCNCPoint3[15288] = {X 230.7574, Y 11.9749, Z -4.6667, A 0.000, B 0.000, C 0.000 }
gfCNCPoint3[15289] = {X 230.7597, Y 12.0808, Z -4.6667, A 0.000, B 0.000, C 0.000 }
gfCNCPoint3[15290] = {X 230.7605, Y 12.1868, Z -4.6667, A 0.000, B 0.000, C 0.000 }
gfCNCPoint3[15291] = {X 230.7602, Y 13.0462, Z -4.6667, A 0.000, B 0.000, C 0.000 }
gfCNCPoint3[15292] = {X 230.6531, Y 14.2235, Z -4.6667, A 0.000, B 0.000, C 0.000 }
gfCNCPoint3[15293] = {X 230.3570, Y 15.3680, Z -4.6667, A 0.000, B 0.000, C 0.000 }
gfCNCPoint3[15294] = {X 229.8795, Y 16.4494, Z -4.6667, A 0.000, B 0.000, C 0.000 }
gfCNCPoint3[15295] = {X 229.2333, Y 17.4394, Z -4.6667, A 0.000, B 0.000, C 0.000 }
gfCNCPoint3[15296] = {X 229.2336, Y 25.8512, Z -4.6667, A 0.000, B 0.000, C 0.000 }
gfCNCPoint3[15297] = {X 231.6336, Y 25.8511, Z -4.6667, A 0.000, B 0.000, C 0.000 }
gfCNCPoint3[15298] = {X 231.6341, Y 38.9914, Z -4.6667, A 0.000, B 0.000, C 0.000 }
gfCNCPoint3[15299] = {X 231.6440, Y 39.0069, Z -4.6667, A 0.000, B 0.000, C 0.000 }
gfCNCPoint3[15300] = {X 232.3931, Y 37.9855, Z -4.6667, A 0.000, B 0.000, C 0.000 }
gfCNCPoint3[15301] = {X 233.2692, Y 37.0706, Z -4.6667, A 0.000, B 0.000, C 0.000 }
gfCNCPoint3[15302] = {X 234.2573, Y 36.2780, Z -4.6667, A 0.000, B 0.000, C 0.000 }
gfCNCPoint3[15303] = {X 235.5693, Y 33.7099, Z -4.6667, A 0.000, B 0.000, C 0.000 }
gfCNCPoint3[15304] = {X 234.4285, Y 32.2857, Z -4.6667, A 0.000, B 0.000, C 0.000 }
gfCNCPoint3[15305] = {X 233.4501, Y 30.7453, Z -4.6667, A 0.000, B 0.000, C 0.000 }
gfCNCPoint3[15306] = {X 232.6459, Y 29.1072, Z -4.6667, A 0.000, B 0.000, C 0.000 }
gfCNCPoint3[15307] = {X 232.0255, Y 27.3911, Z -4.6667, A 0.000, B 0.000, C 0.000 }
gfCNCPoint3[15308] = {X 231.8156, Y 26.6247, Z -4.6667, A 0.000, B 0.000, C 0.000 }
gfCNCPoint3[15309] = {X 231.6336, Y 25.8511, Z -4.6667, A 0.000, B 0.000, C 0.000 }
gfCNCPoint3[15310] = {X 229.2336, Y 25.8512, Z -4.6667, A 0.000, B 0.000, C 0.000 }
gfCNCPoint3[15311] = {X 229.2341, Y 39.7485, Z -4.6667, A 0.000, B 0.000, C 0.000 }
gfCNCPoint3[15312] = {X 229.4334, Y 40.0181, Z -4.6667, A 0.000, B 0.000, C 0.000 }
gfCNCPoint3[15313] = {X 229.6200, Y 40.2966, Z -4.6667, A 0.000, B 0.000, C 0.000 }
gfCNCPoint3[15314] = {X 230.1055, Y 41.1910, Z -4.6667, A 0.000, B 0.000, C 0.000 }
gfCNCPoint3[15315] = {X 230.4616, Y 42.1443, Z -4.6667, A 0.000, B 0.000, C 0.000 }
gfCNCPoint3[15316] = {X 230.6813, Y 43.1379, Z -4.6667, A 0.000, B 0.000, C 0.000 }
gfCNCPoint3[15317] = {X 230.7603, Y 44.1524, Z -4.6667, A 0.000, B 0.000, C 0.000 }
gfCNCPoint3[15318] = {X 230.7605, Y 45.0000, Z -4.6667, A 0.000, B 0.000, C 0.000 }
gfCNCPoint3[15319] = {X 230.7459, Y 45.4609, Z -4.6667, A 0.000, B 0.000, C 0.000 }
gfCNCPoint3[15320] = {X 230.7021, Y 45.9200, Z -4.6667, A 0.000, B 0.000, C 0.000 }
gfCNCPoint3[15321] = {X 232.5859, Y 45.9200, Z -4.6667, A 0.000, B 0.000, C 0.000 }
gfCNCPoint3[15322] = {X 232.5421, Y 45.4609, Z -4.6667, A 0.000, B 0.000, C 0.000 }
gfCNCPoint3[15323] = {X 232.5275, Y 45.0000, Z -4.6667, A 0.000, B 0.000, C 0.000 }
gfCNCPoint3[15324] = {X 232.5275, Y 44.2090, Z -4.6667, A 0.000, B 0.000, C 0.000 }
gfCNCPoint3[15325] = {X 232.6006, Y 43.1798, Z -4.6667, A 0.000, B 0.000, C 0.000 }
gfCNCPoint3[15326] = {X 232.8184, Y 42.1714, Z -4.6667, A 0.000, B 0.000, C 0.000 }
gfCNCPoint3[15327] = {X 233.1766, Y 41.2038, Z -4.6667, A 0.000, B 0.000, C 0.000 }
gfCNCPoint3[15328] = {X 233.6680, Y 40.2966, Z -4.6667, A 0.000, B 0.000, C 0.000 }
gfCNCPoint3[15329] = {X 234.3527, Y 39.3876, Z -4.6667, A 0.000, B 0.000, C 0.000 }
gfCNCPoint3[15330] = {X 235.1707, Y 38.5964, Z -4.6667, A 0.000, B 0.000, C 0.000 }
gfCNCPoint3[15331] = {X 236.1021, Y 37.9424, Z -4.6667, A 0.000, B 0.000, C 0.000 }
gfCNCPoint3[15332] = {X 238.4999, Y 33.2489, Z -4.6667, A 0.000, B 0.000, C 0.000 }
gfCNCPoint3[15333] = {X 237.3861, Y 32.1411, Z -4.6667, A 0.000, B 0.000, C 0.000 }
gfCNCPoint3[15334] = {X 236.4008, Y 30.9176, Z -4.6667, A 0.000, B 0.000, C 0.000 }
gfCNCPoint3[15335] = {X 235.5558, Y 29.5934, Z -4.6667, A 0.000, B 0.000, C 0.000 }
gfCNCPoint3[15336] = {X 234.8614, Y 28.1843, Z -4.6667, A 0.000, B 0.000, C 0.000 }
gfCNCPoint3[15337] = {X 234.3260, Y 26.7074, Z -4.6667, A 0.000, B 0.000, C 0.000 }
gfCNCPoint3[15338] = {X 234.1404, Y 26.0289, Z -4.6667, A 0.000, B 0.000, C 0.000 }
gfCNCPoint3[15339] = {X 233.9794, Y 25.3440, Z -4.6667, A 0.000, B 0.000, C 0.000 }
gfCNCPoint3[15340] = {X 233.6674, Y 23.4555, Z -4.6667, A 0.000, B 0.000, C 0.000 }
gfCNCPoint3[15341] = {X 233.5420, Y 21.5454, Z -4.6667, A 0.000, B 0.000, C 0.000 }
gfCNCPoint3[15342] = {X 233.6046, Y 19.6322, Z -4.6667, A 0.000, B 0.000, C 0.000 }
gfCNCPoint3[15343] = {X 233.8545, Y 17.7344, Z -4.6667, A 0.000, B 0.000, C 0.000 }
gfCNCPoint3[15344] = {X 234.2893, Y 15.8703, Z -4.6667, A 0.000, B 0.000, C 0.000 }
gfCNCPoint3[15345] = {X 234.7353, Y 14.5426, Z -4.6667, A 0.000, B 0.000, C 0.000 }
gfCNCPoint3[15346] = {X 235.3046, Y 13.2630, Z -4.6667, A 0.000, B 0.000, C 0.000 }
gfCNCPoint3[15347] = {X 235.3660, Y 13.1423, Z -4.6667, A 0.000, B 0.000, C 0.000 }
gfCNCPoint3[15348] = {X 235.4285, Y 13.0222, Z -4.6667, A 0.000, B 0.000, C 0.000 }
gfCNCPoint3[15349] = {X 236.1698, Y 11.7671, Z -4.6667, A 0.000, B 0.000, C 0.000 }
gfCNCPoint3[15350] = {X 237.0309, Y 10.5908, Z -4.6667, A 0.000, B 0.000, C 0.000 }
gfCNCPoint3[15351] = {X 238.0035, Y 9.5050, Z -4.6667, A 0.000, B 0.000, C 0.000 }
gfCNCPoint3[15352] = {X 233.3044, Y 9.5050, Z -4.6667, A 0.000, B 0.000, C 0.000 }
gfCNCPoint3[15353] = {X 233.3044, Y 7.1050, Z -4.6667, A 0.000, B 0.000, C 0.000 }
gfCNCPoint3[15354] = {X 191.1448, Y 7.1050, Z -4.6667, A 0.000, B 0.000, C 0.000 }
gfCNCPoint3[15355] = {X 193.1017, Y 7.6482, Z -4.6667, A 0.000, B 0.000, C 0.000 }
gfCNCPoint3[15356] = {X 194.9849, Y 8.4083, Z -4.6667, A 0.000, B 0.000, C 0.000 }
gfCNCPoint3[15357] = {X 196.7706, Y 9.3758, Z -4.6667, A 0.000, B 0.000, C 0.000 }
gfCNCPoint3[15358] = {X 198.4359, Y 10.5382, Z -4.6667, A 0.000, B 0.000, C 0.000 }
gfCNCPoint3[15359] = {X 198.8585, Y 10.8887, Z -4.6667, A 0.000, B 0.000, C 0.000 }
gfCNCPoint3[15360] = {X 199.2666, Y 11.2560, Z -4.6667, A 0.000, B 0.000, C 0.000 }
gfCNCPoint3[15361] = {X 200.3517, Y 12.3984, Z -4.6667, A 0.000, B 0.000, C 0.000 }
gfCNCPoint3[15362] = {X 201.2972, Y 13.6587, Z -4.6667, A 0.000, B 0.000, C 0.000 }
gfCNCPoint3[15363] = {X 202.0904, Y 15.0201, Z -4.6667, A 0.000, B 0.000, C 0.000 }
gfCNCPoint3[15364] = {X 202.7207, Y 16.4641, Z -4.6667, A 0.000, B 0.000, C 0.000 }
gfCNCPoint3[15365] = {X 203.2143, Y 18.1838, Z -4.6667, A 0.000, B 0.000, C 0.000 }
gfCNCPoint3[15366] = {X 203.5076, Y 19.9487, Z -4.6667, A 0.000, B 0.000, C 0.000 }
gfCNCPoint3[15367] = {X 203.5967, Y 21.7356, Z -4.6667, A 0.000, B 0.000, C 0.000 }
gfCNCPoint3[15368] = {X 203.4803, Y 23.5210, Z -4.6667, A 0.000, B 0.000, C 0.000 }
gfCNCPoint3[15369] = {X 203.1601, Y 25.2812, Z -4.6667, A 0.000, B 0.000, C 0.000 }
gfCNCPoint3[15370] = {X 202.7597, Y 26.6266, Z -4.6667, A 0.000, B 0.000, C 0.000 }
gfCNCPoint3[15371] = {X 202.2081, Y 27.9173, Z -4.6667, A 0.000, B 0.000, C 0.000 }
gfCNCPoint3[15372] = {X 201.5124, Y 29.1365, Z -4.6667, A 0.000, B 0.000, C 0.000 }
gfCNCPoint3[15373] = {X 200.6819, Y 30.2682, Z -4.6667, A 0.000, B 0.000, C 0.000 }
gfCNCPoint3[15374] = {X 199.7275, Y 31.2974, Z -4.6667, A 0.000, B 0.000, C 0.000 }
gfCNCPoint3[15375] = {X 200.5669, Y 31.8699, Z -4.6667, A 0.000, B 0.000, C 0.000 }
gfCNCPoint3[15376] = {X 201.2695, Y 32.6038, Z -4.6667, A 0.000, B 0.000, C 0.000 }
gfCNCPoint3[15377] = {X 201.8050, Y 33.4673, Z -4.6667, A 0.000, B 0.000, C 0.000 }
gfCNCPoint3[15378] = {X 204.8262, Y 39.7091, Z -4.6667, A 0.000, B 0.000, C 0.000 }
gfCNCPoint3[15379] = {X 205.1508, Y 40.5847, Z -4.6667, A 0.000, B 0.000, C 0.000 }
gfCNCPoint3[15380] = {X 205.3026, Y 41.5062, Z -4.6667, A 0.000, B 0.000, C 0.000 }
gfCNCPoint3[15381] = {X 205.2761, Y 42.4397, Z -4.6667, A 0.000, B 0.000, C 0.000 }
gfCNCPoint3[15382] = {X 205.0723, Y 43.3511, Z -4.6667, A 0.000, B 0.000, C 0.000 }
gfCNCPoint3[15383] = {X 204.6986, Y 44.2070, Z -4.6667, A 0.000, B 0.000, C 0.000 }
gfCNCPoint3[15384] = {X 204.1687, Y 44.9760, Z -4.6667, A 0.000, B 0.000, C 0.000 }
gfCNCPoint3[15385] = {X 203.5020, Y 45.6299, Z -4.6667, A 0.000, B 0.000, C 0.000 }
gfCNCPoint3[15386] = {X 202.9657, Y 46.0635, Z -4.6667, A 0.000, B 0.000, C 0.000 }
gfCNCPoint3[15387] = {X 202.2137, Y 46.5640, Z -4.6667, A 0.000, B 0.000, C 0.000 }
gfCNCPoint3[15388] = {X 201.3825, Y 46.9177, Z -4.6667, A 0.000, B 0.000, C 0.000 }
gfCNCPoint3[15389] = {X 200.5004, Y 47.1126, Z -4.6667, A 0.000, B 0.000, C 0.000 }
gfCNCPoint3[15390] = {X 199.5976, Y 47.1420, Z -4.6667, A 0.000, B 0.000, C 0.000 }
gfCNCPoint3[15391] = {X 198.7047, Y 47.0048, Z -4.6667, A 0.000, B 0.000, C 0.000 }
gfCNCPoint3[15392] = {X 196.3904, Y 48.1794, Z -4.6667, A 0.000, B 0.000, C 0.000 }
gfCNCPoint3[15393] = {X 193.9811, Y 49.1442, Z -4.6667, A 0.000, B 0.000, C 0.000 }
gfCNCPoint3[15394] = {X 191.4958, Y 49.8916, Z -4.6667, A 0.000, B 0.000, C 0.000 }
gfCNCPoint3[15395] = {X 190.2926, Y 50.1572, Z -4.6667, A 0.000, B 0.000, C 0.000 }
gfCNCPoint3[15396] = {X 189.0770, Y 50.3586, Z -4.6667, A 0.000, B 0.000, C 0.000 }
gfCNCPoint3[15397] = {X 186.8988, Y 50.5562, Z -4.6667, A 0.000, B 0.000, C 0.000 }
gfCNCPoint3[15398] = {X 184.7116, Y 50.5479, Z -4.6667, A 0.000, B 0.000, C 0.000 }
gfCNCPoint3[15399] = {X 184.7360, Y 50.0685, Z -4.6667, A 0.000, B 0.000, C 0.000 }
gfCNCPoint3[15400] = {X 183.1155, Y 49.9277, Z -4.6667, A 0.000, B 0.000, C 0.000 }
gfCNCPoint3[15401] = {X 181.5093, Y 49.6713, Z -4.6667, A 0.000, B 0.000, C 0.000 }
gfCNCPoint3[15402] = {X 179.6141, Y 49.1975, Z -4.6667, A 0.000, B 0.000, C 0.000 }
gfCNCPoint3[15403] = {X 177.7853, Y 48.5109, Z -4.6667, A 0.000, B 0.000, C 0.000 }
gfCNCPoint3[15404] = {X 176.0466, Y 47.6203, Z -4.6667, A 0.000, B 0.000, C 0.000 }
gfCNCPoint3[15405] = {X 174.4208, Y 46.5375, Z -4.6667, A 0.000, B 0.000, C 0.000 }
gfCNCPoint3[15406] = {X 173.1806, Y 45.4907, Z -4.6667, A 0.000, B 0.000, C 0.000 }
gfCNCPoint3[15407] = {X 172.0769, Y 44.3009, Z -4.6667, A 0.000, B 0.000, C 0.000 }
gfCNCPoint3[15408] = {X 171.1262, Y 42.9857, Z -4.6667, A 0.000, B 0.000, C 0.000 }
gfCNCPoint3[15409] = {X 170.3426, Y 41.5646, Z -4.6667, A 0.000, B 0.000, C 0.000 }
gfCNCPoint3[15410] = {X 169.7376, Y 40.0587, Z -4.6667, A 0.000, B 0.000, C 0.000 }
gfCNCPoint3[15411] = {X 169.3203, Y 38.4904, Z -4.6667, A 0.000, B 0.000, C 0.000 }
gfCNCPoint3[15412] = {X 169.0969, Y 36.8830, Z -4.6667, A 0.000, B 0.000, C 0.000 }
gfCNCPoint3[15413] = {X 169.0127, Y 35.0392, Z -4.6667, A 0.000, B 0.000, C 0.000 }
gfCNCPoint3[15414] = {X 169.1599, Y 33.1994, Z -4.6667, A 0.000, B 0.000, C 0.000 }
gfCNCPoint3[15415] = {X 169.5362, Y 31.3925, Z -4.6667, A 0.000, B 0.000, C 0.000 }
gfCNCPoint3[15416] = {X 170.1356, Y 29.6468, Z -4.6667, A 0.000, B 0.000, C 0.000 }
gfCNCPoint3[15417] = {X 170.7626, Y 28.3592, Z -4.6667, A 0.000, B 0.000, C 0.000 }
gfCNCPoint3[15418] = {X 171.5525, Y 27.1646, Z -4.6667, A 0.000, B 0.000, C 0.000 }
gfCNCPoint3[15419] = {X 172.4916, Y 26.0833, Z -4.6667, A 0.000, B 0.000, C 0.000 }
gfCNCPoint3[15420] = {X 173.5640, Y 25.1341, Z -4.6667, A 0.000, B 0.000, C 0.000 }
gfCNCPoint3[15421] = {X 174.7511, Y 24.3330, Z -4.6667, A 0.000, B 0.000, C 0.000 }
gfCNCPoint3[15422] = {X 173.9911, Y 23.9227, Z -4.6667, A 0.000, B 0.000, C 0.000 }
gfCNCPoint3[15423] = {X 173.3258, Y 23.3718, Z -4.6667, A 0.000, B 0.000, C 0.000 }
gfCNCPoint3[15424] = {X 172.7810, Y 22.7016, Z -4.6667, A 0.000, B 0.000, C 0.000 }
gfCNCPoint3[15425] = {X 172.3776, Y 21.9378, Z -4.6667, A 0.000, B 0.000, C 0.000 }
gfCNCPoint3[15426] = {X 169.7664, Y 15.5423, Z -4.6667, A 0.000, B 0.000, C 0.000 }
gfCNCPoint3[15427] = {X 169.5126, Y 14.6752, Z -4.6667, A 0.000, B 0.000, C 0.000 }
gfCNCPoint3[15428] = {X 169.4412, Y 13.7745, Z -4.6667, A 0.000, B 0.000, C 0.000 }
gfCNCPoint3[15429] = {X 169.5553, Y 12.8782, Z -4.6667, A 0.000, B 0.000, C 0.000 }
gfCNCPoint3[15430] = {X 169.8501, Y 12.0242, Z -4.6667, A 0.000, B 0.000, C 0.000 }
gfCNCPoint3[15431] = {X 170.3131, Y 11.2483, Z -4.6667, A 0.000, B 0.000, C 0.000 }
gfCNCPoint3[15432] = {X 170.9248, Y 10.5834, Z -4.6667, A 0.000, B 0.000, C 0.000 }
gfCNCPoint3[15433] = {X 171.6594, Y 10.0574, Z -4.6667, A 0.000, B 0.000, C 0.000 }
gfCNCPoint3[15434] = {X 172.2916, Y 9.6970, Z -4.6667, A 0.000, B 0.000, C 0.000 }
gfCNCPoint3[15435] = {X 173.1812, Y 9.3215, Z -4.6667, A 0.000, B 0.000, C 0.000 }
gfCNCPoint3[15436] = {X 174.1312, Y 9.1491, Z -4.6667, A 0.000, B 0.000, C 0.000 }
gfCNCPoint3[15437] = {X 175.0959, Y 9.1881, Z -4.6667, A 0.000, B 0.000, C 0.000 }
gfCNCPoint3[15438] = {X 176.0289, Y 9.4365, Z -4.6667, A 0.000, B 0.000, C 0.000 }
gfCNCPoint3[15439] = {X 178.2247, Y 8.5149, Z -4.6667, A 0.000, B 0.000, C 0.000 }
gfCNCPoint3[15440] = {X 180.5016, Y 7.8175, Z -4.6667, A 0.000, B 0.000, C 0.000 }
gfCNCPoint3[15441] = {X 182.8368, Y 7.3511, Z -4.6667, A 0.000, B 0.000, C 0.000 }
gfCNCPoint3[15442] = {X 185.2069, Y 7.1204, Z -4.6667, A 0.000, B 0.000, C 0.000 }
gfCNCPoint3[15443] = {X 187.5882, Y 7.1278, Z -4.6667, A 0.000, B 0.000, C 0.000 }
gfCNCPoint3[15444] = {X 189.9568, Y 7.3732, Z -4.6667, A 0.000, B 0.000, C 0.000 }
gfCNCPoint3[15445] = {X 191.7228, Y 7.7363, Z -4.6667, A 0.000, B 0.000, C 0.000 }
gfCNCPoint3[15446] = {X 193.4421, Y 8.2789, Z -4.6667, A 0.000, B 0.000, C 0.000 }
gfCNCPoint3[15447] = {X 195.0965, Y 8.9953, Z -4.6667, A 0.000, B 0.000, C 0.000 }
gfCNCPoint3[15448] = {X 196.6685, Y 9.8779, Z -4.6667, A 0.000, B 0.000, C 0.000 }
gfCNCPoint3[15449] = {X 198.1416, Y 10.9173, Z -4.6667, A 0.000, B 0.000, C 0.000 }
gfCNCPoint3[15450] = {X 199.2084, Y 11.8667, Z -4.6667, A 0.000, B 0.000, C 0.000 }
gfCNCPoint3[15451] = {X 200.1655, Y 12.9264, Z -4.6667, A 0.000, B 0.000, C 0.000 }
gfCNCPoint3[15452] = {X 201.0016, Y 14.0840, Z -4.6667, A 0.000, B 0.000, C 0.000 }
gfCNCPoint3[15453] = {X 201.7068, Y 15.3258, Z -4.6667, A 0.000, B 0.000, C 0.000 }
gfCNCPoint3[15454] = {X 202.2727, Y 16.6369, Z -4.6667, A 0.000, B 0.000, C 0.000 }
gfCNCPoint3[15455] = {X 202.7489, Y 18.3014, Z -4.6667, A 0.000, B 0.000, C 0.000 }
gfCNCPoint3[15456] = {X 203.0315, Y 20.0095, Z -4.6667, A 0.000, B 0.000, C 0.000 }
gfCNCPoint3[15457] = {X 203.1167, Y 21.7387, Z -4.6667, A 0.000, B 0.000, C 0.000 }
gfCNCPoint3[15458] = {X 203.0035, Y 23.4663, Z -4.6667, A 0.000, B 0.000, C 0.000 }
gfCNCPoint3[15459] = {X 202.6933, Y 25.1696, Z -4.6667, A 0.000, B 0.000, C 0.000 }
gfCNCPoint3[15460] = {X 202.2585, Y 26.5986, Z -4.6667, A 0.000, B 0.000, C 0.000 }
gfCNCPoint3[15461] = {X 201.6464, Y 27.9610, Z -4.6667, A 0.000, B 0.000, C 0.000 }
gfCNCPoint3[15462] = {X 200.8667, Y 29.2350, Z -4.6667, A 0.000, B 0.000, C 0.000 }
gfCNCPoint3[15463] = {X 199.9319, Y 30.4001, Z -4.6667, A 0.000, B 0.000, C 0.000 }
gfCNCPoint3[15464] = {X 198.8572, Y 31.4373, Z -4.6667, A 0.000, B 0.000, C 0.000 }
gfCNCPoint3[15465] = {X 199.6403, Y 31.7991, Z -4.6667, A 0.000, B 0.000, C 0.000 }
gfCNCPoint3[15466] = {X 200.3378, Y 32.3067, Z -4.6667, A 0.000, B 0.000, C 0.000 }
gfCNCPoint3[15467] = {X 200.9228, Y 32.9406, Z -4.6667, A 0.000, B 0.000, C 0.000 }
gfCNCPoint3[15468] = {X 201.3730, Y 33.6764, Z -4.6667, A 0.000, B 0.000, C 0.000 }
gfCNCPoint3[15469] = {X 204.3942, Y 39.9182, Z -4.6667, A 0.000, B 0.000, C 0.000 }
gfCNCPoint3[15470] = {X 204.7207, Y 40.8441, Z -4.6667, A 0.000, B 0.000, C 0.000 }
gfCNCPoint3[15471] = {X 204.8337, Y 41.8194, Z -4.6667, A 0.000, B 0.000, C 0.000 }
gfCNCPoint3[15472] = {X 204.7276, Y 42.7955, Z -4.6667, A 0.000, B 0.000, C 0.000 }
gfCNCPoint3[15473] = {X 204.4078, Y 43.7238, Z -4.6667, A 0.000, B 0.000, C 0.000 }
gfCNCPoint3[15474] = {X 203.8900, Y 44.5580, Z -4.6667, A 0.000, B 0.000, C 0.000 }
gfCNCPoint3[15475] = {X 203.2002, Y 45.2567, Z -4.6667, A 0.000, B 0.000, C 0.000 }
gfCNCPoint3[15476] = {X 202.6640, Y 45.6902, Z -4.6667, A 0.000, B 0.000, C 0.000 }
gfCNCPoint3[15477] = {X 201.9525, Y 46.1594, Z -4.6667, A 0.000, B 0.000, C 0.000 }
gfCNCPoint3[15478] = {X 201.1642, Y 46.4830, Z -4.6667, A 0.000, B 0.000, C 0.000 }
gfCNCPoint3[15479] = {X 200.3283, Y 46.6490, Z -4.6667, A 0.000, B 0.000, C 0.000 }
gfCNCPoint3[15480] = {X 199.4762, Y 46.6513, Z -4.6667, A 0.000, B 0.000, C 0.000 }
gfCNCPoint3[15481] = {X 198.6395, Y 46.4897, Z -4.6667, A 0.000, B 0.000, C 0.000 }
gfCNCPoint3[15482] = {X 196.3111, Y 47.6881, Z -4.6667, A 0.000, B 0.000, C 0.000 }
gfCNCPoint3[15483] = {X 193.8834, Y 48.6698, Z -4.6667, A 0.000, B 0.000, C 0.000 }
gfCNCPoint3[15484] = {X 191.3765, Y 49.4267, Z -4.6667, A 0.000, B 0.000, C 0.000 }
gfCNCPoint3[15485] = {X 189.1876, Y 49.8580, Z -4.6667, A 0.000, B 0.000, C 0.000 }
gfCNCPoint3[15486] = {X 186.9670, Y 50.0726, Z -4.6667, A 0.000, B 0.000, C 0.000 }
gfCNCPoint3[15487] = {X 184.7360, Y 50.0685, Z -4.6667, A 0.000, B 0.000, C 0.000 }
gfCNCPoint3[15488] = {X 184.7116, Y 50.5479, Z -4.6667, A 0.000, B 0.000, C 0.000 }
gfCNCPoint3[15489] = {X 185.7077, Y 51.5013, Z -4.6667, A 0.000, B 0.000, C 0.000 }
gfCNCPoint3[15490] = {X 186.5583, Y 52.5866, Z -4.6667, A 0.000, B 0.000, C 0.000 }
gfCNCPoint3[15491] = {X 187.2461, Y 53.7818, Z -4.6667, A 0.000, B 0.000, C 0.000 }
gfCNCPoint3[15492] = {X 187.7795, Y 55.1339, Z -4.6667, A 0.000, B 0.000, C 0.000 }
gfCNCPoint3[15493] = {X 188.1044, Y 56.5506, Z -4.6667, A 0.000, B 0.000, C 0.000 }
gfCNCPoint3[15494] = {X 188.2135, Y 58.0000, Z -4.6667, A 0.000, B 0.000, C 0.000 }
gfCNCPoint3[15495] = {X 188.2132, Y 59.0140, Z -4.6667, A 0.000, B 0.000, C 0.000 }
gfCNCPoint3[15496] = {X 188.2026, Y 59.3926, Z -4.6667, A 0.000, B 0.000, C 0.000 }
gfCNCPoint3[15497] = {X 188.1773, Y 59.7704, Z -4.6667, A 0.000, B 0.000, C 0.000 }
gfCNCPoint3[15498] = {X 206.8561, Y 80.1560, Z -4.6667, A 0.000, B 0.000, C 0.000 }
gfCNCPoint3[15499] = {X 212.1646, Y 75.2919, Z -4.6667, A 0.000, B 0.000, C 0.000 }
gfCNCPoint3[15500] = {X 215.1994, Y 78.6039, Z -4.6667, A 0.000, B 0.000, C 0.000 }
gfCNCPoint3[15501] = {X 218.3274, Y 76.6000, Z -4.6667, A 0.000, B 0.000, C 0.000 }
gfCNCPoint3[15502] = {X 216.9968, Y 76.0778, Z -4.6667, A 0.000, B 0.000, C 0.000 }
gfCNCPoint3[15503] = {X 216.3757, Y 75.8850, Z -4.6667, A 0.000, B 0.000, C 0.000 }
gfCNCPoint3[15504] = {X 215.7306, Y 75.8034, Z -4.6667, A 0.000, B 0.000, C 0.000 }
gfCNCPoint3[15505] = {X 213.9339, Y 75.6430, Z -4.6667, A 0.000, B 0.000, C 0.000 }
gfCNCPoint3[15506] = {X 212.1646, Y 75.2919, Z -4.6667, A 0.000, B 0.000, C 0.000 }
gfCNCPoint3[15507] = {X 210.3951, Y 76.9132, Z -4.6667, A 0.000, B 0.000, C 0.000 }
gfCNCPoint3[15508] = {X 214.7939, Y 81.7140, Z -4.6667, A 0.000, B 0.000, C 0.000 }
gfCNCPoint3[15509] = {X 223.5821, Y 76.0839, Z -4.6667, A 0.000, B 0.000, C 0.000 }
gfCNCPoint3[15510] = {X 217.8859, Y 73.8485, Z -4.6667, A 0.000, B 0.000, C 0.000 }
gfCNCPoint3[15511] = {X 216.8716, Y 73.5368, Z -4.6667, A 0.000, B 0.000, C 0.000 }
gfCNCPoint3[15512] = {X 215.8187, Y 73.4050, Z -4.6667, A 0.000, B 0.000, C 0.000 }
gfCNCPoint3[15513] = {X 214.2761, Y 73.2675, Z -4.6667, A 0.000, B 0.000, C 0.000 }
gfCNCPoint3[15514] = {X 212.7570, Y 72.9661, Z -4.6667, A 0.000, B 0.000, C 0.000 }
gfCNCPoint3[15515] = {X 211.1578, Y 72.4585, Z -4.6667, A 0.000, B 0.000, C 0.000 }
gfCNCPoint3[15516] = {X 209.6281, Y 71.7693, Z -4.6667, A 0.000, B 0.000, C 0.000 }
gfCNCPoint3[15517] = {X 208.1884, Y 70.9078, Z -4.6667, A 0.000, B 0.000, C 0.000 }
gfCNCPoint3[15518] = {X 206.8580, Y 69.8856, Z -4.6667, A 0.000, B 0.000, C 0.000 }
gfCNCPoint3[15519] = {X 205.6547, Y 68.7163, Z -4.6667, A 0.000, B 0.000, C 0.000 }
gfCNCPoint3[15520] = {X 204.5948, Y 67.4157, Z -4.6667, A 0.000, B 0.000, C 0.000 }
gfCNCPoint3[15521] = {X 203.6925, Y 66.0012, Z -4.6667, A 0.000, B 0.000, C 0.000 }
gfCNCPoint3[15522] = {X 202.9599, Y 64.4918, Z -4.6667, A 0.000, B 0.000, C 0.000 }
gfCNCPoint3[15523] = {X 202.4067, Y 62.9078, Z -4.6667, A 0.000, B 0.000, C 0.000 }
gfCNCPoint3[15524] = {X 202.0405, Y 61.2705, Z -4.6667, A 0.000, B 0.000, C 0.000 }
gfCNCPoint3[15525] = {X 199.6720, Y 61.6577, Z -4.6667, A 0.000, B 0.000, C 0.000 }
gfCNCPoint3[15526] = {X 199.5094, Y 60.3400, Z -4.6667, A 0.000, B 0.000, C 0.000 }
gfCNCPoint3[15527] = {X 199.4510, Y 59.0136, Z -4.6667, A 0.000, B 0.000, C 0.000 }
gfCNCPoint3[15528] = {X 199.4508, Y 58.0000, Z -4.6667, A 0.000, B 0.000, C 0.000 }
gfCNCPoint3[15529] = {X 199.5412, Y 56.2559, Z -4.6667, A 0.000, B 0.000, C 0.000 }
gfCNCPoint3[15530] = {X 199.8112, Y 54.5304, Z -4.6667, A 0.000, B 0.000, C 0.000 }
gfCNCPoint3[15531] = {X 197.5977, Y 55.4815, Z -4.6667, A 0.000, B 0.000, C 0.000 }
gfCNCPoint3[15532] = {X 195.3261, Y 56.2843, Z -4.6667, A 0.000, B 0.000, C 0.000 }
gfCNCPoint3[15533] = {X 195.3578, Y 56.6300, Z -4.6667, A 0.000, B 0.000, C 0.000 }
gfCNCPoint3[15534] = {X 195.3824, Y 56.9762, Z -4.6667, A 0.000, B 0.000, C 0.000 }
gfCNCPoint3[15535] = {X 199.6720, Y 61.6577, Z -4.6667, A 0.000, B 0.000, C 0.000 }
gfCNCPoint3[15536] = {X 202.0405, Y 61.2705, Z -4.6667, A 0.000, B 0.000, C 0.000 }
gfCNCPoint3[15537] = {X 201.9013, Y 60.1426, Z -4.6667, A 0.000, B 0.000, C 0.000 }
gfCNCPoint3[15538] = {X 201.8510, Y 59.0073, Z -4.6667, A 0.000, B 0.000, C 0.000 }
gfCNCPoint3[15539] = {X 201.8508, Y 58.0000, Z -4.6667, A 0.000, B 0.000, C 0.000 }
gfCNCPoint3[15540] = {X 201.9283, Y 56.5038, Z -4.6667, A 0.000, B 0.000, C 0.000 }
gfCNCPoint3[15541] = {X 202.1600, Y 55.0237, Z -4.6667, A 0.000, B 0.000, C 0.000 }
gfCNCPoint3[15542] = {X 202.4967, Y 53.7235, Z -4.6667, A 0.000, B 0.000, C 0.000 }
gfCNCPoint3[15543] = {X 202.9525, Y 52.4600, Z -4.6667, A 0.000, B 0.000, C 0.000 }
gfCNCPoint3[15544] = {X 203.5234, Y 51.2442, Z -4.6667, A 0.000, B 0.000, C 0.000 }
gfCNCPoint3[15545] = {X 202.2636, Y 51.6558, Z -4.6667, A 0.000, B 0.000, C 0.000 }
gfCNCPoint3[15546] = {X 200.9595, Y 51.8916, Z -4.6667, A 0.000, B 0.000, C 0.000 }
gfCNCPoint3[15547] = {X 199.6354, Y 51.9474, Z -4.6667, A 0.000, B 0.000, C 0.000 }
gfCNCPoint3[15548] = {X 199.2148, Y 52.1555, Z -4.6667, A 0.000, B 0.000, C 0.000 }
gfCNCPoint3[15549] = {X 198.7914, Y 52.3578, Z -4.6667, A 0.000, B 0.000, C 0.000 }
gfCNCPoint3[15550] = {X 196.7764, Y 53.2256, Z -4.6667, A 0.000, B 0.000, C 0.000 }
gfCNCPoint3[15551] = {X 194.7096, Y 53.9617, Z -4.6667, A 0.000, B 0.000, C 0.000 }
gfCNCPoint3[15552] = {X 192.5997, Y 54.5632, Z -4.6667, A 0.000, B 0.000, C 0.000 }
gfCNCPoint3[15553] = {X 192.9063, Y 56.2411, Z -4.6667, A 0.000, B 0.000, C 0.000 }
gfCNCPoint3[15554] = {X 193.0134, Y 57.9433, Z -4.6667, A 0.000, B 0.000, C 0.000 }
gfCNCPoint3[15555] = {X 210.3951, Y 76.9132, Z -4.6667, A 0.000, B 0.000, C 0.000 }
gfCNCPoint3[15556] = {X 208.6256, Y 78.5346, Z -4.6667, A 0.000, B 0.000, C 0.000 }
gfCNCPoint3[15557] = {X 214.3884, Y 84.8240, Z -4.6667, A 0.000, B 0.000, C 0.000 }
gfCNCPoint3[15558] = {X 228.8368, Y 75.5678, Z -4.6667, A 0.000, B 0.000, C 0.000 }
gfCNCPoint3[15559] = {X 218.7729, Y 71.6185, Z -4.6667, A 0.000, B 0.000, C 0.000 }
gfCNCPoint3[15560] = {X 217.8430, Y 71.3045, Z -4.6667, A 0.000, B 0.000, C 0.000 }
gfCNCPoint3[15561] = {X 216.8831, Y 71.0997, Z -4.6667, A 0.000, B 0.000, C 0.000 }
gfCNCPoint3[15562] = {X 215.9060, Y 71.0066, Z -4.6667, A 0.000, B 0.000, C 0.000 }
gfCNCPoint3[15563] = {X 214.2362, Y 70.8311, Z -4.6667, A 0.000, B 0.000, C 0.000 }
gfCNCPoint3[15564] = {X 212.6069, Y 70.4258, Z -4.6667, A 0.000, B 0.000, C 0.000 }
gfCNCPoint3[15565] = {X 211.0495, Y 69.7984, Z -4.6667, A 0.000, B 0.000, C 0.000 }
gfCNCPoint3[15566] = {X 209.5941, Y 68.9612, Z -4.6667, A 0.000, B 0.000, C 0.000 }
gfCNCPoint3[15567] = {X 208.2689, Y 67.9303, Z -4.6667, A 0.000, B 0.000, C 0.000 }
gfCNCPoint3[15568] = {X 207.0994, Y 66.7256, Z -4.6667, A 0.000, B 0.000, C 0.000 }
gfCNCPoint3[15569] = {X 206.1082, Y 65.3703, Z -4.6667, A 0.000, B 0.000, C 0.000 }
gfCNCPoint3[15570] = {X 205.3146, Y 63.8908, Z -4.6667, A 0.000, B 0.000, C 0.000 }
gfCNCPoint3[15571] = {X 204.7337, Y 62.3154, Z -4.6667, A 0.000, B 0.000, C 0.000 }
gfCNCPoint3[15572] = {X 204.3769, Y 60.6748, Z -4.6667, A 0.000, B 0.000, C 0.000 }
gfCNCPoint3[15573] = {X 204.2510, Y 59.0005, Z -4.6667, A 0.000, B 0.000, C 0.000 }
gfCNCPoint3[15574] = {X 204.2508, Y 58.0000, Z -4.6667, A 0.000, B 0.000, C 0.000 }
gfCNCPoint3[15575] = {X 204.3396, Y 56.5377, Z -4.6667, A 0.000, B 0.000, C 0.000 }
gfCNCPoint3[15576] = {X 204.6048, Y 55.0969, Z -4.6667, A 0.000, B 0.000, C 0.000 }
gfCNCPoint3[15577] = {X 205.0425, Y 53.6988, Z -4.6667, A 0.000, B 0.000, C 0.000 }
gfCNCPoint3[15578] = {X 205.6462, Y 52.3639, Z -4.6667, A 0.000, B 0.000, C 0.000 }
gfCNCPoint3[15579] = {X 206.5297, Y 50.9385, Z -4.6667, A 0.000, B 0.000, C 0.000 }
gfCNCPoint3[15580] = {X 207.6021, Y 49.6492, Z -4.6667, A 0.000, B 0.000, C 0.000 }
gfCNCPoint3[15581] = {X 208.8427, Y 48.5208, Z -4.6667, A 0.000, B 0.000, C 0.000 }
gfCNCPoint3[15582] = {X 210.2277, Y 47.5751, Z -4.6667, A 0.000, B 0.000, C 0.000 }
gfCNCPoint3[15583] = {X 209.8801, Y 46.3328, Z -4.6667, A 0.000, B 0.000, C 0.000 }
gfCNCPoint3[15584] = {X 209.7572, Y 45.0487, Z -4.6667, A 0.000, B 0.000, C 0.000 }
gfCNCPoint3[15585] = {X 209.7570, Y 44.1958, Z -4.6667, A 0.000, B 0.000, C 0.000 }
gfCNCPoint3[15586] = {X 209.8559, Y 43.0060, Z -4.6667, A 0.000, B 0.000, C 0.000 }
gfCNCPoint3[15587] = {X 210.1497, Y 41.8488, Z -4.6667, A 0.000, B 0.000, C 0.000 }
gfCNCPoint3[15588] = {X 210.6304, Y 40.7559, Z -4.6667, A 0.000, B 0.000, C 0.000 }
gfCNCPoint3[15589] = {X 211.2849, Y 39.7574, Z -4.6667, A 0.000, B 0.000, C 0.000 }
gfCNCPoint3[15590] = {X 211.2849, Y 37.0768, Z -4.6667, A 0.000, B 0.000, C 0.000 }
gfCNCPoint3[15591] = {X 208.8849, Y 37.0768, Z -4.6667, A 0.000, B 0.000, C 0.000 }
gfCNCPoint3[15592] = {X 208.8849, Y 18.1977, Z -4.6667, A 0.000, B 0.000, C 0.000 }
gfCNCPoint3[15593] = {X 208.2329, Y 17.0017, Z -4.6667, A 0.000, B 0.000, C 0.000 }
gfCNCPoint3[15594] = {X 207.7553, Y 15.7260, Z -4.6667, A 0.000, B 0.000, C 0.000 }
gfCNCPoint3[15595] = {X 207.4614, Y 14.3959, Z -4.6667, A 0.000, B 0.000, C 0.000 }
gfCNCPoint3[15596] = {X 207.3572, Y 13.0378, Z -4.6667, A 0.000, B 0.000, C 0.000 }
gfCNCPoint3[15597] = {X 207.3570, Y 12.1868, Z -4.6667, A 0.000, B 0.000, C 0.000 }
gfCNCPoint3[15598] = {X 207.3580, Y 12.0459, Z -4.6667, A 0.000, B 0.000, C 0.000 }
gfCNCPoint3[15599] = {X 207.3611, Y 11.9050, Z -4.6667, A 0.000, B 0.000, C 0.000 }
gfCNCPoint3[15600] = {X 205.8572, Y 11.9050, Z -4.6667, A 0.000, B 0.000, C 0.000 }
gfCNCPoint3[15601] = {X 206.6123, Y 13.3419, Z -4.6667, A 0.000, B 0.000, C 0.000 }
gfCNCPoint3[15602] = {X 207.2377, Y 14.8398, Z -4.6667, A 0.000, B 0.000, C 0.000 }
gfCNCPoint3[15603] = {X 207.7984, Y 16.7126, Z -4.6667, A 0.000, B 0.000, C 0.000 }
gfCNCPoint3[15604] = {X 208.1772, Y 18.6305, Z -4.6667, A 0.000, B 0.000, C 0.000 }
gfCNCPoint3[15605] = {X 208.3705, Y 20.5758, Z -4.6667, A 0.000, B 0.000, C 0.000 }
gfCNCPoint3[15606] = {X 208.3766, Y 22.5308, Z -4.6667, A 0.000, B 0.000, C 0.000 }
gfCNCPoint3[15607] = {X 208.1954, Y 24.4773, Z -4.6667, A 0.000, B 0.000, C 0.000 }
gfCNCPoint3[15608] = {X 207.8285, Y 26.3975, Z -4.6667, A 0.000, B 0.000, C 0.000 }
gfCNCPoint3[15609] = {X 207.3614, Y 28.0099, Z -4.6667, A 0.000, B 0.000, C 0.000 }
gfCNCPoint3[15610] = {X 206.7381, Y 29.5686, Z -4.6667, A 0.000, B 0.000, C 0.000 }
gfCNCPoint3[15611] = {X 205.9645, Y 31.0584, Z -4.6667, A 0.000, B 0.000, C 0.000 }
gfCNCPoint3[15612] = {X 206.0465, Y 31.2165, Z -4.6667, A 0.000, B 0.000, C 0.000 }
gfCNCPoint3[15613] = {X 206.1255, Y 31.3760, Z -4.6667, A 0.000, B 0.000, C 0.000 }
gfCNCPoint3[15614] = {X 208.8849, Y 37.0768, Z -4.6667, A 0.000, B 0.000, C 0.000 }
gfCNCPoint3[15615] = {X 211.2849, Y 37.0768, Z -4.6667, A 0.000, B 0.000, C 0.000 }
gfCNCPoint3[15616] = {X 211.2846, Y 17.4399, Z -4.6667, A 0.000, B 0.000, C 0.000 }
gfCNCPoint3[15617] = {X 210.6362, Y 16.4461, Z -4.6667, A 0.000, B 0.000, C 0.000 }
gfCNCPoint3[15618] = {X 210.1578, Y 15.3602, Z -4.6667, A 0.000, B 0.000, C 0.000 }
gfCNCPoint3[15619] = {X 209.8622, Y 14.2110, Z -4.6667, A 0.000, B 0.000, C 0.000 }
gfCNCPoint3[15620] = {X 209.7572, Y 13.0291, Z -4.6667, A 0.000, B 0.000, C 0.000 }
gfCNCPoint3[15621] = {X 209.7570, Y 12.1868, Z -4.6667, A 0.000, B 0.000, C 0.000 }
gfCNCPoint3[15622] = {X 209.7578, Y 12.0808, Z -4.6667, A 0.000, B 0.000, C 0.000 }
gfCNCPoint3[15623] = {X 209.7601, Y 11.9749, Z -4.6667, A 0.000, B 0.000, C 0.000 }
gfCNCPoint3[15624] = {X 209.9068, Y 10.7177, Z -4.6667, A 0.000, B 0.000, C 0.000 }
gfCNCPoint3[15625] = {X 210.2690, Y 9.5050, Z -4.6667, A 0.000, B 0.000, C 0.000 }
gfCNCPoint3[15626] = {X 200.9079, Y 9.5050, Z -4.6667, A 0.000, B 0.000, C 0.000 }
gfCNCPoint3[15627] = {X 201.9815, Y 10.6134, Z -4.6667, A 0.000, B 0.000, C 0.000 }
gfCNCPoint3[15628] = {X 202.9432, Y 11.8202, Z -4.6667, A 0.000, B 0.000, C 0.000 }
gfCNCPoint3[15629] = {X 203.7840, Y 13.1141, Z -4.6667, A 0.000, B 0.000, C 0.000 }
gfCNCPoint3[15630] = {X 204.4374, Y 14.3567, Z -4.6667, A 0.000, B 0.000, C 0.000 }
gfCNCPoint3[15631] = {X 204.9792, Y 15.6519, Z -4.6667, A 0.000, B 0.000, C 0.000 }
gfCNCPoint3[15632] = {X 205.5516, Y 17.6384, Z -4.6667, A 0.000, B 0.000, C 0.000 }
gfCNCPoint3[15633] = {X 205.8923, Y 19.6774, Z -4.6667, A 0.000, B 0.000, C 0.000 }
gfCNCPoint3[15634] = {X 205.9967, Y 21.7421, Z -4.6667, A 0.000, B 0.000, C 0.000 }
gfCNCPoint3[15635] = {X 205.8635, Y 23.8052, Z -4.6667, A 0.000, B 0.000, C 0.000 }
gfCNCPoint3[15636] = {X 205.4943, Y 25.8393, Z -4.6667, A 0.000, B 0.000, C 0.000 }
gfCNCPoint3[15637] = {X 205.0932, Y 27.2255, Z -4.6667, A 0.000, B 0.000, C 0.000 }
gfCNCPoint3[15638] = {X 204.5577, Y 28.5656, Z -4.6667, A 0.000, B 0.000, C 0.000 }
gfCNCPoint3[15639] = {X 203.8929, Y 29.8465, Z -4.6667, A 0.000, B 0.000, C 0.000 }
gfCNCPoint3[15640] = {X 203.1054, Y 31.0559, Z -4.6667, A 0.000, B 0.000, C 0.000 }
gfCNCPoint3[15641] = {X 203.5733, Y 31.7149, Z -4.6667, A 0.000, B 0.000, C 0.000 }
